LIN {X 0,Y 523.515,Z 618.573,A -85,B 0,C 180,E1 -4762.285,E2 -4762.285} C_VEL
LIN {X 0,Y 523.436,Z 624.082,A -85,B 0,C 180,E1 -4763.834,E2 -4763.834} C_VEL
LIN {X 0,Y 523.322,Z 628.245,A -85,B 0,C 180,E1 -4765.378,E2 -4765.378} C_VEL
LIN {X 0,Y 523.358,Z 631.166,A -85,B 0,C 180,E1 -4766.921,E2 -4766.921} C_VEL
LIN {X 0,Y 523.272,Z 632.904,A -85,B 0,C 180,E1 -4768.461,E2 -4768.461} C_VEL
LIN {X 0,Y 523.243,Z 633.498,A -85,B 0,C 180,E1 -4770,E2 -4770} C_VEL
LIN {X 0,Y 523.272,Z 632.901,A -85,B 0,C 180,E1 -4771.539,E2 -4771.539} C_VEL
LIN {X 0,Y 523.358,Z 631.161,A -85,B 0,C 180,E1 -4773.079,E2 -4773.079} C_VEL
LIN {X 0,Y 523.322,Z 628.242,A -85,B 0,C 180,E1 -4774.622,E2 -4774.622} C_VEL
LIN {X 0,Y 523.43,Z 624.086,A -85,B 0,C 180,E1 -4776.166,E2 -4776.166} C_VEL
LIN {X 0,Y 523.515,Z 618.574,A -85,B 0,C 180,E1 -4777.715,E2 -4777.715} C_VEL
LIN {X 0,Y 523.699,Z 611.561,A -85,B 0,C 180,E1 -4779.267,E2 -4779.267} C_VEL
LIN {X 0,Y 523.951,Z 602.835,A -85,B 0,C 180,E1 -4780.823,E2 -4780.823} C_VEL
LIN {X 0,Y 524.214,Z 593.543,A -85,B 0,C 180,E1 -4782.193,E2 -4782.193} C_VEL
LIN {X 0,Y 524.552,Z 584.141,A -85,B 0,C 180,E1 -4783.362,E2 -4783.362} C_VEL
LIN {X 0,Y 524.988,Z 571.926,A -85,B 0,C 180,E1 -4784.636,E2 -4784.636} C_VEL
LIN {X 0,Y 525.434,Z 560.572,A -85,B 0,C 180,E1 -4785.625,E2 -4785.625} C_VEL
LIN {X 0,Y 525.869,Z 547.217,A -85,B 0,C 180,E1 -4786.598,E2 -4786.598} C_VEL
LIN {X 0,Y 526.404,Z 533.994,A -85,B 0,C 180,E1 -4787.381,E2 -4787.381} C_VEL
LIN {X 0,Y 526.831,Z 519.537,A -85,B 0,C 180,E1 -4788.068,E2 -4788.068} C_VEL
LIN {X 0,Y 527.21,Z 505.352,A -85,B 0,C 180,E1 -4788.583,E2 -4788.583} C_VEL
LIN {X 0,Y 527.474,Z 490.49,A -85,B 0,C 180,E1 -4788.97,E2 -4788.97} C_VEL
LIN {X 0,Y 527.688,Z 469.477,A -85,B 0,C 180,E1 -4789.303,E2 -4789.303} C_VEL
LIN {X 0,Y 528.493,Z 334.8,A -85,B 0,C 180,E1 -4791.181,E2 -4791.181} C_VEL
LIN {X 0,Y 525.743,Z 320.905,A -85,B 0,C 180,E1 -4791.506,E2 -4791.506} C_VEL
LIN {X 0,Y 526.391,Z 301.543,A -85,B 0,C 180,E1 -4794.029,E2 -4794.029} C_VEL
LIN {X 0,Y 526.808,Z 285.78,A -85,B 0,C 180,E1 -4796.119,E2 -4796.119} C_VEL
LIN {X 0,Y 523.953,Z 272.848,A -85,B 0,C 180,E1 -4798.053,E2 -4798.053} C_VEL
LIN {X 0,Y 523.94,Z 272.843,A -85,B 0,C 180,E1 -4800.854,E2 -4800.854} C_VEL
LIN {X 0,Y 523.953,Z 272.844,A -85,B 0,C 180,E1 -4803.733,E2 -4803.733} C_VEL
LIN {X 0,Y 523.883,Z 272.854,A -85,B 0,C 180,E1 -4806.398,E2 -4806.398} C_VEL
LIN {X 0,Y 523.905,Z 272.847,A -85,B 0,C 180,E1 -4809.085,E2 -4809.085} C_VEL
LIN {X 0,Y 523.892,Z 272.856,A -85,B 0,C 180,E1 -4812.123,E2 -4812.123} C_VEL
LIN {X 0,Y 523.927,Z 272.844,A -85,B 0,C 180,E1 -4815.31,E2 -4815.31} C_VEL
LIN {X 0,Y 523.914,Z 272.845,A -85,B 0,C 180,E1 -4818.693,E2 -4818.693} C_VEL
LIN {X 0,Y 523.891,Z 272.854,A -85,B 0,C 180,E1 -4821.896,E2 -4821.896} C_VEL
LIN {X 0,Y 523.906,Z 272.844,A -85,B 0,C 180,E1 -4824.912,E2 -4824.912} C_VEL
LIN {X 0,Y 523.923,Z 272.849,A -85,B 0,C 180,E1 -4827.679,E2 -4827.679} C_VEL
LIN {X 0,Y 523.939,Z 272.841,A -85,B 0,C 180,E1 -4830.677,E2 -4830.677} C_VEL
LIN {X 0,Y 523.878,Z 272.856,A -85,B 0,C 180,E1 -4833.723,E2 -4833.723} C_VEL
LIN {X 0,Y 523.895,Z 272.848,A -85,B 0,C 180,E1 -4836.269,E2 -4836.269} C_VEL
LIN {X 0,Y 523.931,Z 272.842,A -85,B 0,C 180,E1 -4838.766,E2 -4838.766} C_VEL
LIN {X 0,Y 523.919,Z 272.84,A -85,B 0,C 180,E1 -4841.22,E2 -4841.22} C_VEL
LIN {X 0,Y 523.89,Z 272.855,A -85,B 0,C 180,E1 -4843.637,E2 -4843.637} C_VEL
LIN {X 0,Y 523.901,Z 272.846,A -85,B 0,C 180,E1 -4846.027,E2 -4846.027} C_VEL
LIN {X 0,Y 523.942,Z 272.83,A -85,B 0,C 180,E1 -4848.393,E2 -4848.393} C_VEL
LIN {X 0,Y 523.931,Z 272.85,A -85,B 0,C 180,E1 -4851.515,E2 -4851.515} C_VEL
LIN {X 0,Y 523.998,Z 272.835,A -85,B 0,C 180,E1 -4853.84,E2 -4853.84} C_VEL
LIN {X 0,Y 524.012,Z 272.835,A -85,B 0,C 180,E1 -4856.925,E2 -4856.925} C_VEL
LIN {X 0,Y 524.106,Z 272.825,A -85,B 0,C 180,E1 -4859.232,E2 -4859.232} C_VEL
LIN {X 0,Y 524.086,Z 272.821,A -85,B 0,C 180,E1 -4862.306,E2 -4862.306} C_VEL
LIN {X 0,Y 524.051,Z 272.834,A -85,B 0,C 180,E1 -4865.387,E2 -4865.387} C_VEL
LIN {X 0,Y 523.991,Z 272.838,A -85,B 0,C 180,E1 -4867.708,E2 -4867.708} C_VEL
LIN {X 0,Y 523.972,Z 272.839,A -85,B 0,C 180,E1 -4870.823,E2 -4870.823} C_VEL
LIN {X 0,Y 523.925,Z 272.852,A -85,B 0,C 180,E1 -4873.182,E2 -4873.182} C_VEL
LIN {X 0,Y 523.92,Z 272.847,A -85,B 0,C 180,E1 -4875.562,E2 -4875.562} C_VEL
LIN {X 0,Y 523.932,Z 272.841,A -85,B 0,C 180,E1 -4877.97,E2 -4877.97} C_VEL
LIN {X 0,Y 523.945,Z 272.834,A -85,B 0,C 180,E1 -4880.411,E2 -4880.411} C_VEL
LIN {X 0,Y 523.895,Z 272.85,A -85,B 0,C 180,E1 -4882.894,E2 -4882.894} C_VEL
LIN {X 0,Y 523.902,Z 272.847,A -85,B 0,C 180,E1 -4885.421,E2 -4885.421} C_VEL
LIN {X 0,Y 523.946,Z 272.835,A -85,B 0,C 180,E1 -4888,E2 -4888} C_VEL
LIN {X 0,Y 523.929,Z 272.85,A -85,B 0,C 180,E1 -4890.854,E2 -4890.854} C_VEL
LIN {X 0,Y 523.92,Z 272.844,A -85,B 0,C 180,E1 -4893.73,E2 -4893.73} C_VEL
LIN {X 0,Y 523.894,Z 272.849,A -85,B 0,C 180,E1 -4896.402,E2 -4896.402} C_VEL
LIN {X 0,Y 523.91,Z 272.849,A -85,B 0,C 180,E1 -4899.086,E2 -4899.086} C_VEL
LIN {X 0,Y 523.944,Z 272.841,A -85,B 0,C 180,E1 -4902.12,E2 -4902.12} C_VEL
LIN {X 0,Y 523.935,Z 272.844,A -85,B 0,C 180,E1 -4905.311,E2 -4905.311} C_VEL
LIN {X 0,Y 523.909,Z 272.852,A -85,B 0,C 180,E1 -4906.876,E2 -4906.876} C_VEL
LIN {X 0,Y 523.234,Z 272.932,A -85,B 0,C 180,E1 -4907.518,E2 -4907.518} C_VEL
LIN {X 0,Y 520.367,Z 273.294,A -85,B 0,C 180,E1 -4908.559,E2 -4908.559} C_VEL
LIN {X 0,Y 517.961,Z 273.589,A -85,B 0,C 180,E1 -4909.398,E2 -4909.398} C_VEL
LIN {X 0,Y 516.948,Z 273.715,A -85,B 0,C 180,E1 -4910.046,E2 -4910.046} C_VEL
LIN {X 0,Y 516.876,Z 273.725,A -85,B 0,C 180,E1 -4910.265,E2 -4910.265} C_VEL
LIN {X 0,Y 516.873,Z 273.722,A -85,B 0,C 180,E1 -4913.344,E2 -4913.344} C_VEL
LIN {X 0,Y 516.882,Z 273.724,A -85,B 0,C 180,E1 -4916.12,E2 -4916.12} C_VEL
LIN {X 0,Y 516.889,Z 273.725,A -85,B 0,C 180,E1 -4918.937,E2 -4918.937} C_VEL
LIN {X 0,Y 516.909,Z 273.72,A -85,B 0,C 180,E1 -4921.585,E2 -4921.585} C_VEL
LIN {X 0,Y 516.909,Z 273.725,A -85,B 0,C 180,E1 -4924.642,E2 -4924.642} C_VEL
LIN {X 0,Y 516.953,Z 273.863,A -85,B 0,C 180,E1 -4924.967,E2 -4924.967} C_VEL
LIN {X 0,Y 519.043,Z 283.843,A -85,B 0,C 180,E1 -4926.669,E2 -4926.669} C_VEL
LIN {X 0,Y 518.916,Z 294.305,A -85,B 0,C 180,E1 -4928.269,E2 -4928.269} C_VEL
LIN {X 0,Y 521.961,Z 307.972,A -85,B 0,C 180,E1 -4928.603,E2 -4928.603} C_VEL
LIN {X 0,Y 521.148,Z 429.496,A -85,B 0,C 180,E1 -4930.322,E2 -4930.322} C_VEL
LIN {X 0,Y 520.872,Z 460.237,A -85,B 0,C 180,E1 -4930.782,E2 -4930.782} C_VEL
LIN {X 0,Y 520.583,Z 475.638,A -85,B 0,C 180,E1 -4931.172,E2 -4931.172} C_VEL
LIN {X 0,Y 520.26,Z 490.103,A -85,B 0,C 180,E1 -4931.696,E2 -4931.696} C_VEL
LIN {X 0,Y 519.79,Z 502.789,A -85,B 0,C 180,E1 -4932.289,E2 -4932.289} C_VEL
LIN {X 0,Y 519.276,Z 516.39,A -85,B 0,C 180,E1 -4933.084,E2 -4933.084} C_VEL
LIN {X 0,Y 518.746,Z 529.412,A -85,B 0,C 180,E1 -4934.017,E2 -4934.017} C_VEL
LIN {X 0,Y 518.235,Z 541.543,A -85,B 0,C 180,E1 -4935.069,E2 -4935.069} C_VEL
LIN {X 0,Y 517.757,Z 553.011,A -85,B 0,C 180,E1 -4936.259,E2 -4936.259} C_VEL
LIN {X 0,Y 517.338,Z 562.659,A -85,B 0,C 180,E1 -4937.446,E2 -4937.446} C_VEL
LIN {X 0,Y 517.02,Z 572.112,A -85,B 0,C 180,E1 -4938.831,E2 -4938.831} C_VEL
LIN {X 0,Y 516.736,Z 579.983,A -85,B 0,C 180,E1 -4940.212,E2 -4940.212} C_VEL
LIN {X 0,Y 516.528,Z 587.329,A -85,B 0,C 180,E1 -4941.787,E2 -4941.787} C_VEL
LIN {X 0,Y 516.408,Z 591.836,A -85,B 0,C 180,E1 -4942.965,E2 -4942.965} C_VEL
LIN {X 0,Y 516.377,Z 596.61,A -85,B 0,C 180,E1 -4944.533,E2 -4944.533} C_VEL
LIN {X 0,Y 516.326,Z 600.112,A -85,B 0,C 180,E1 -4946.098,E2 -4946.098} C_VEL
LIN {X 0,Y 516.258,Z 602.432,A -85,B 0,C 180,E1 -4947.659,E2 -4947.659} C_VEL
LIN {X 0,Y 516.156,Z 603.623,A -85,B 0,C 180,E1 -4949.22,E2 -4949.22} C_VEL
LIN {X 0,Y 516.157,Z 603.642,A -85,B 0,C 180,E1 -4950.78,E2 -4950.78} C_VEL
LIN {X 0,Y 516.259,Z 602.527,A -85,B 0,C 180,E1 -4952.341,E2 -4952.341} C_VEL
LIN {X 0,Y 516.326,Z 600.282,A -85,B 0,C 180,E1 -4953.902,E2 -4953.902} C_VEL
LIN {X 0,Y 516.373,Z 596.852,A -85,B 0,C 180,E1 -4955.467,E2 -4955.467} C_VEL
LIN {X 0,Y 516.407,Z 592.155,A -85,B 0,C 180,E1 -4957.035,E2 -4957.035} C_VEL
LIN {X 0,Y 516.573,Z 586.066,A -85,B 0,C 180,E1 -4958.607,E2 -4958.607} C_VEL
LIN {X 0,Y 516.762,Z 578.399,A -85,B 0,C 180,E1 -4960.183,E2 -4960.183} C_VEL
LIN {X 0,Y 517.051,Z 570.22,A -85,B 0,C 180,E1 -4961.565,E2 -4961.565} C_VEL
LIN {X 0,Y 517.442,Z 560.368,A -85,B 0,C 180,E1 -4962.95,E2 -4962.95} C_VEL
LIN {X 0,Y 517.879,Z 550.263,A -85,B 0,C 180,E1 -4964.138,E2 -4964.138} C_VEL
LIN {X 0,Y 518.346,Z 538.482,A -85,B 0,C 180,E1 -4965.307,E2 -4965.307} C_VEL
LIN {X 0,Y 518.956,Z 525.014,A -85,B 0,C 180,E1 -4966.411,E2 -4966.411} C_VEL
LIN {X 0,Y 519.551,Z 511.488,A -85,B 0,C 180,E1 -4967.313,E2 -4967.313} C_VEL
LIN {X 0,Y 519.966,Z 497.613,A -85,B 0,C 180,E1 -4968.06,E2 -4968.06} C_VEL
LIN {X 0,Y 520.423,Z 483.39,A -85,B 0,C 180,E1 -4968.655,E2 -4968.655} C_VEL
LIN {X 0,Y 520.729,Z 468.583,A -85,B 0,C 180,E1 -4969.116,E2 -4969.116} C_VEL
LIN {X 0,Y 520.978,Z 453.076,A -85,B 0,C 180,E1 -4969.432,E2 -4969.432} C_VEL
LIN {X 0,Y 521.996,Z 308.384,A -85,B 0,C 180,E1 -4971.48,E2 -4971.48} C_VEL
LIN {X 0,Y 518.876,Z 293.935,A -85,B 0,C 180,E1 -4971.852,E2 -4971.852} C_VEL
LIN {X 0,Y 519.153,Z 284.409,A -85,B 0,C 180,E1 -4973.326,E2 -4973.326} C_VEL
LIN {X 0,Y 516.923,Z 273.723,A -85,B 0,C 180,E1 -4975.169,E2 -4975.169} C_VEL
LIN {X 0,Y 516.917,Z 273.723,A -85,B 0,C 180,E1 -4977.903,E2 -4977.903} C_VEL
LIN {X 0,Y 516.889,Z 273.723,A -85,B 0,C 180,E1 -4980.203,E2 -4980.203} C_VEL
LIN {X 0,Y 516.892,Z 273.724,A -85,B 0,C 180,E1 -4982.946,E2 -4982.946} C_VEL
LIN {X 0,Y 516.885,Z 273.727,A -85,B 0,C 180,E1 -4985.778,E2 -4985.778} C_VEL
LIN {X 0,Y 516.876,Z 273.725,A -85,B 0,C 180,E1 -4988.715,E2 -4988.715} C_VEL
LIN {X 0,Y 516.906,Z 273.722,A -85,B 0,C 180,E1 -4991.774,E2 -4991.774} C_VEL
LIN {X 0,Y 516.889,Z 273.725,A -85,B 0,C 180,E1 -4995.006,E2 -4995.006} C_VEL
LIN {X 0,Y 516.906,Z 273.712,A -85,B 0,C 180,E1 -4998.398,E2 -4998.398} C_VEL
LIN {X 0,Y 516.871,Z 273.728,A -85,B 0,C 180,E1 -5001.283,E2 -5001.283} C_VEL
LIN {X 0,Y 516.862,Z 273.719,A -85,B 0,C 180,E1 -5004.219,E2 -5004.219} C_VEL
LIN {X 0,Y 516.871,Z 273.729,A -85,B 0,C 180,E1 -5007.051,E2 -5007.051} C_VEL
LIN {X 0,Y 516.877,Z 273.716,A -85,B 0,C 180,E1 -5009.795,E2 -5009.795} C_VEL
LIN {X 0,Y 516.913,Z 273.718,A -85,B 0,C 180,E1 -5012.466,E2 -5012.466} C_VEL
LIN {X 0,Y 516.844,Z 273.732,A -85,B 0,C 180,E1 -5015.068,E2 -5015.068} C_VEL
LIN {X 0,Y 516.857,Z 273.723,A -85,B 0,C 180,E1 -5017.621,E2 -5017.621} C_VEL
LIN {X 0,Y 516.917,Z 273.716,A -85,B 0,C 180,E1 -5020.129,E2 -5020.129} C_VEL
LIN {X 0,Y 516.885,Z 273.722,A -85,B 0,C 180,E1 -5022.595,E2 -5022.595} C_VEL
LIN {X 0,Y 516.927,Z 273.72,A -85,B 0,C 180,E1 -5025.03,E2 -5025.03} C_VEL
LIN {X 0,Y 516.953,Z 273.712,A -85,B 0,C 180,E1 -5028.233,E2 -5028.233} C_VEL
LIN {X 0,Y 516.938,Z 273.713,A -85,B 0,C 180,E1 -5031.399,E2 -5031.399} C_VEL
LIN {X 0,Y 516.971,Z 273.709,A -85,B 0,C 180,E1 -5033.756,E2 -5033.756} C_VEL
LIN {X 0,Y 516.968,Z 273.716,A -85,B 0,C 180,E1 -5036.883,E2 -5036.883} C_VEL
LIN {X 0,Y 517.074,Z 273.696,A -85,B 0,C 180,E1 -5039.221,E2 -5039.221} C_VEL
LIN {X 0,Y 516.938,Z 273.713,A -85,B 0,C 180,E1 -5041.558,E2 -5041.558} C_VEL
LIN {X 0,Y 516.956,Z 273.713,A -85,B 0,C 180,E1 -5043.117,E2 -5043.117} C_VEL
LIN {X 0,Y 516.968,Z 273.713,A -85,B 0,C 180,E1 -5046.244,E2 -5046.244} C_VEL
LIN {X 0,Y 516.9,Z 273.716,A -85,B 0,C 180,E1 -5049.39,E2 -5049.39} C_VEL
LIN {X 0,Y 516.939,Z 273.715,A -85,B 0,C 180,E1 -5051.807,E2 -5051.807} C_VEL
LIN {X 0,Y 516.931,Z 273.716,A -85,B 0,C 180,E1 -5055.146,E2 -5055.146} C_VEL
LIN {X 0,Y 516.863,Z 273.727,A -85,B 0,C 180,E1 -5058.224,E2 -5058.224} C_VEL
LIN {X 0,Y 516.899,Z 273.722,A -85,B 0,C 180,E1 -5060.702,E2 -5060.702} C_VEL
LIN {X 0,Y 516.871,Z 273.728,A -85,B 0,C 180,E1 -5064.074,E2 -5064.074} C_VEL
LIN {X 0,Y 516.823,Z 273.732,A -85,B 0,C 180,E1 -5066.663,E2 -5066.663} C_VEL
LIN {X 0,Y 516.895,Z 273.72,A -85,B 0,C 180,E1 -5069.523,E2 -5069.523} C_VEL
LIN {X 0,Y 516.883,Z 273.722,A -85,B 0,C 180,E1 -5072.544,E2 -5072.544} C_VEL
LIN {X 0,Y 516.839,Z 273.726,A -85,B 0,C 180,E1 -5075.328,E2 -5075.328} C_VEL
LIN {X 0,Y 516.863,Z 273.723,A -85,B 0,C 180,E1 -5078.717,E2 -5078.717} C_VEL
LIN {X 0,Y 516.875,Z 273.721,A -85,B 0,C 180,E1 -5081.779,E2 -5081.779} C_VEL
LIN {X 0,Y 516.888,Z 273.72,A -85,B 0,C 180,E1 -5085.008,E2 -5085.008} C_VEL
LIN {X 0,Y 516.848,Z 273.728,A -85,B 0,C 180,E1 -5088.407,E2 -5088.407} C_VEL
LIN {X 0,Y 516.867,Z 273.724,A -85,B 0,C 180,E1 -5091.284,E2 -5091.284} C_VEL
LIN {X 0,Y 516.856,Z 273.726,A -85,B 0,C 180,E1 -5094.672,E2 -5094.672} C_VEL
LIN {X 0,Y 516.891,Z 273.725,A -85,B 0,C 180,E1 -5097.458,E2 -5097.458} C_VEL
LIN {X 0,Y 516.917,Z 273.721,A -85,B 0,C 180,E1 -5100.696,E2 -5100.696} C_VEL
LIN {X 0,Y 516.93,Z 273.878,A -85,B 0,C 180,E1 -5101.726,E2 -5101.726} C_VEL
LIN {X 0,Y 519.954,Z 287.167,A -85,B 0,C 180,E1 -5103.727,E2 -5103.727} C_VEL
LIN {X 0,Y 519.424,Z 306.078,A -85,B 0,C 180,E1 -5106.264,E2 -5106.264} C_VEL
LIN {X 0,Y 518.905,Z 320.752,A -85,B 0,C 180,E1 -5108.203,E2 -5108.203} C_VEL
LIN {X 0,Y 521.908,Z 336.644,A -85,B 0,C 180,E1 -5108.568,E2 -5108.568} C_VEL
LIN {X 0,Y 520.848,Z 486.861,A -85,B 0,C 180,E1 -5110.705,E2 -5110.705} C_VEL
LIN {X 0,Y 520.496,Z 502.829,A -85,B 0,C 180,E1 -5111.092,E2 -5111.092} C_VEL
LIN {X 0,Y 520.088,Z 518.191,A -85,B 0,C 180,E1 -5111.638,E2 -5111.638} C_VEL
LIN {X 0,Y 519.608,Z 531.979,A -85,B 0,C 180,E1 -5112.283,E2 -5112.283} C_VEL
LIN {X 0,Y 519.082,Z 545.494,A -85,B 0,C 180,E1 -5113.077,E2 -5113.077} C_VEL
LIN {X 0,Y 518.596,Z 558.466,A -85,B 0,C 180,E1 -5114.011,E2 -5114.011} C_VEL
LIN {X 0,Y 518.028,Z 571.715,A -85,B 0,C 180,E1 -5115.163,E2 -5115.163} C_VEL
LIN {X 0,Y 517.547,Z 583.935,A -85,B 0,C 180,E1 -5116.453,E2 -5116.453} C_VEL
LIN {X 0,Y 517.131,Z 594.805,A -85,B 0,C 180,E1 -5117.84,E2 -5117.84} C_VEL
LIN {X 0,Y 516.883,Z 603.856,A -85,B 0,C 180,E1 -5119.225,E2 -5119.225} C_VEL
LIN {X 0,Y 516.609,Z 611.362,A -85,B 0,C 180,E1 -5120.605,E2 -5120.605} C_VEL
LIN {X 0,Y 516.451,Z 618.369,A -85,B 0,C 180,E1 -5122.179,E2 -5122.179} C_VEL
LIN {X 0,Y 516.356,Z 623.878,A -85,B 0,C 180,E1 -5123.749,E2 -5123.749} C_VEL
LIN {X 0,Y 516.238,Z 628.041,A -85,B 0,C 180,E1 -5125.315,E2 -5125.315} C_VEL
LIN {X 0,Y 516.272,Z 630.963,A -85,B 0,C 180,E1 -5126.879,E2 -5126.879} C_VEL
LIN {X 0,Y 516.189,Z 632.703,A -85,B 0,C 180,E1 -5128.44,E2 -5128.44} C_VEL
LIN {X 0,Y 516.151,Z 633.299,A -85,B 0,C 180,E1 -5130,E2 -5130} C_VEL
LIN {X 0,Y 516.189,Z 632.7,A -85,B 0,C 180,E1 -5131.56,E2 -5131.56} C_VEL
LIN {X 0,Y 516.272,Z 630.958,A -85,B 0,C 180,E1 -5133.121,E2 -5133.121} C_VEL
LIN {X 0,Y 516.238,Z 628.039,A -85,B 0,C 180,E1 -5134.685,E2 -5134.685} C_VEL
LIN {X 0,Y 516.328,Z 623.881,A -85,B 0,C 180,E1 -5136.251,E2 -5136.251} C_VEL
LIN {X 0,Y 516.451,Z 618.37,A -85,B 0,C 180,E1 -5137.821,E2 -5137.821} C_VEL
LIN {X 0,Y 516.609,Z 611.356,A -85,B 0,C 180,E1 -5139.395,E2 -5139.395} C_VEL
LIN {X 0,Y 516.881,Z 603.852,A -85,B 0,C 180,E1 -5140.775,E2 -5140.775} C_VEL
LIN {X 0,Y 517.113,Z 595.075,A -85,B 0,C 180,E1 -5142.121,E2 -5142.121} C_VEL
LIN {X 0,Y 517.497,Z 585.575,A -85,B 0,C 180,E1 -5143.348,E2 -5143.348} C_VEL
LIN {X 0,Y 517.897,Z 574.703,A -85,B 0,C 180,E1 -5144.539,E2 -5144.539} C_VEL
LIN {X 0,Y 518.399,Z 563.427,A -85,B 0,C 180,E1 -5145.581,E2 -5145.581} C_VEL
LIN {X 0,Y 518.906,Z 549.877,A -85,B 0,C 180,E1 -5146.625,E2 -5146.625} C_VEL
LIN {X 0,Y 519.523,Z 535.561,A -85,B 0,C 180,E1 -5147.517,E2 -5147.517} C_VEL
LIN {X 0,Y 519.986,Z 521.595,A -85,B 0,C 180,E1 -5148.213,E2 -5148.213} C_VEL
LIN {X 0,Y 520.413,Z 506.675,A -85,B 0,C 180,E1 -5148.783,E2 -5148.783} C_VEL
LIN {X 0,Y 520.759,Z 491.492,A -85,B 0,C 180,E1 -5149.197,E2 -5149.197} C_VEL
LIN {X 0,Y 520.96,Z 472.786,A -85,B 0,C 180,E1 -5149.512,E2 -5149.512} C_VEL
LIN {X 0,Y 521.866,Z 335.88,A -85,B 0,C 180,E1 -5151.445,E2 -5151.445} C_VEL
LIN {X 0,Y 518.899,Z 320.738,A -85,B 0,C 180,E1 -5151.798,E2 -5151.798} C_VEL
LIN {X 0,Y 519.608,Z 299.781,A -85,B 0,C 180,E1 -5154.576,E2 -5154.576} C_VEL
LIN {X 0,Y 519.962,Z 287.167,A -85,B 0,C 180,E1 -5156.273,E2 -5156.273} C_VEL
LIN {X 0,Y 516.889,Z 273.728,A -85,B 0,C 180,E1 -5158.312,E2 -5158.312} C_VEL
LIN {X 0,Y 516.885,Z 273.721,A -85,B 0,C 180,E1 -5161.109,E2 -5161.109} C_VEL
LIN {X 0,Y 516.901,Z 273.724,A -85,B 0,C 180,E1 -5163.965,E2 -5163.965} C_VEL
LIN {X 0,Y 516.838,Z 273.729,A -85,B 0,C 180,E1 -5166.748,E2 -5166.748} C_VEL
LIN {X 0,Y 516.851,Z 273.73,A -85,B 0,C 180,E1 -5169.723,E2 -5169.723} C_VEL
LIN {X 0,Y 516.835,Z 273.728,A -85,B 0,C 180,E1 -5172.835,E2 -5172.835} C_VEL
LIN {X 0,Y 516.887,Z 273.72,A -85,B 0,C 180,E1 -5175.006,E2 -5175.006} C_VEL
LIN {X 0,Y 516.878,Z 273.724,A -85,B 0,C 180,E1 -5178.401,E2 -5178.401} C_VEL
LIN {X 0,Y 516.863,Z 273.724,A -85,B 0,C 180,E1 -5181.283,E2 -5181.283} C_VEL
LIN {X 0,Y 516.842,Z 273.725,A -85,B 0,C 180,E1 -5184.672,E2 -5184.672} C_VEL
LIN {X 0,Y 516.883,Z 273.723,A -85,B 0,C 180,E1 -5187.456,E2 -5187.456} C_VEL
LIN {X 0,Y 516.907,Z 273.717,A -85,B 0,C 180,E1 -5190.695,E2 -5190.695} C_VEL
LIN {X 0,Y 516.856,Z 273.732,A -85,B 0,C 180,E1 -5193.82,E2 -5193.82} C_VEL
LIN {X 0,Y 516.844,Z 273.724,A -85,B 0,C 180,E1 -5196.775,E2 -5196.775} C_VEL
LIN {X 0,Y 516.926,Z 273.716,A -85,B 0,C 180,E1 -5199.732,E2 -5199.732} C_VEL
LIN {X 0,Y 516.87,Z 273.719,A -85,B 0,C 180,E1 -5202.594,E2 -5202.594} C_VEL
LIN {X 0,Y 516.918,Z 273.718,A -85,B 0,C 180,E1 -5205.029,E2 -5205.029} C_VEL
LIN {X 0,Y 516.911,Z 273.706,A -85,B 0,C 180,E1 -5208.233,E2 -5208.233} C_VEL
LIN {X 0,Y 516.904,Z 273.723,A -85,B 0,C 180,E1 -5211.399,E2 -5211.399} C_VEL
LIN {X 0,Y 516.967,Z 273.712,A -85,B 0,C 180,E1 -5213.756,E2 -5213.756} C_VEL
LIN {X 0,Y 516.953,Z 273.714,A -85,B 0,C 180,E1 -5216.883,E2 -5216.883} C_VEL
LIN {X 0,Y 517.077,Z 273.7,A -85,B 0,C 180,E1 -5219.221,E2 -5219.221} C_VEL
LIN {X 0,Y 517.058,Z 273.696,A -85,B 0,C 180,E1 -5222.337,E2 -5222.337} C_VEL
LIN {X 0,Y 516.998,Z 273.711,A -85,B 0,C 180,E1 -5225.46,E2 -5225.46} C_VEL
LIN {X 0,Y 516.947,Z 273.714,A -85,B 0,C 180,E1 -5227.814,E2 -5227.814} C_VEL
LIN {X 0,Y 516.93,Z 273.718,A -85,B 0,C 180,E1 -5230.973,E2 -5230.973} C_VEL
LIN {X 0,Y 516.885,Z 273.726,A -85,B 0,C 180,E1 -5233.365,E2 -5233.365} C_VEL
LIN {X 0,Y 516.881,Z 273.722,A -85,B 0,C 180,E1 -5235.78,E2 -5235.78} C_VEL
LIN {X 0,Y 516.9,Z 273.717,A -85,B 0,C 180,E1 -5238.223,E2 -5238.223} C_VEL
LIN {X 0,Y 516.892,Z 273.715,A -85,B 0,C 180,E1 -5240.702,E2 -5240.702} C_VEL
LIN {X 0,Y 516.874,Z 273.721,A -85,B 0,C 180,E1 -5244.074,E2 -5244.074} C_VEL
LIN {X 0,Y 516.896,Z 273.72,A -85,B 0,C 180,E1 -5246.659,E2 -5246.659} C_VEL
LIN {X 0,Y 516.898,Z 273.72,A -85,B 0,C 180,E1 -5249.524,E2 -5249.524} C_VEL
LIN {X 0,Y 516.884,Z 273.722,A -85,B 0,C 180,E1 -5252.544,E2 -5252.544} C_VEL
LIN {X 0,Y 516.856,Z 273.726,A -85,B 0,C 180,E1 -5255.33,E2 -5255.33} C_VEL
LIN {X 0,Y 516.87,Z 273.721,A -85,B 0,C 180,E1 -5257.944,E2 -5257.944} C_VEL
LIN {X 0,Y 516.875,Z 273.727,A -85,B 0,C 180,E1 -5260.743,E2 -5260.743} C_VEL
LIN {X 0,Y 516.875,Z 273.728,A -85,B 0,C 180,E1 -5262.832,E2 -5262.832} C_VEL
LIN {X 0,Y 516.889,Z 273.726,A -85,B 0,C 180,E1 -5265.008,E2 -5265.008} C_VEL
LIN {X 0,Y 516.907,Z 273.722,A -85,B 0,C 180,E1 -5268.4,E2 -5268.4} C_VEL
LIN {X 0,Y 516.876,Z 273.725,A -85,B 0,C 180,E1 -5270.265,E2 -5270.265} C_VEL
LIN {X 0,Y 516.239,Z 273.809,A -85,B 0,C 180,E1 -5270.915,E2 -5270.915} C_VEL
LIN {X 0,Y 513.396,Z 274.163,A -85,B 0,C 180,E1 -5271.97,E2 -5271.97} C_VEL
LIN {X 0,Y 510.967,Z 274.464,A -85,B 0,C 180,E1 -5272.82,E2 -5272.82} C_VEL
LIN {X 0,Y 509.91,Z 274.59,A -85,B 0,C 180,E1 -5273.477,E2 -5273.477} C_VEL
LIN {X 0,Y 509.818,Z 274.6,A -85,B 0,C 180,E1 -5273.699,E2 -5273.699} C_VEL
LIN {X 0,Y 509.839,Z 274.603,A -85,B 0,C 180,E1 -5276.539,E2 -5276.539} C_VEL
LIN {X 0,Y 509.843,Z 274.6,A -85,B 0,C 180,E1 -5279.335,E2 -5279.335} C_VEL
LIN {X 0,Y 509.885,Z 274.598,A -85,B 0,C 180,E1 -5282.055,E2 -5282.055} C_VEL
LIN {X 0,Y 509.898,Z 274.718,A -85,B 0,C 180,E1 -5284.706,E2 -5284.706} C_VEL
LIN {X 0,Y 512.177,Z 285.37,A -85,B 0,C 180,E1 -5286.552,E2 -5286.552} C_VEL
LIN {X 0,Y 512.032,Z 294.252,A -85,B 0,C 180,E1 -5287.951,E2 -5287.951} C_VEL
LIN {X 0,Y 515.351,Z 308.882,A -85,B 0,C 180,E1 -5288.324,E2 -5288.324} C_VEL
LIN {X 0,Y 514.53,Z 420.915,A -85,B 0,C 180,E1 -5289.93,E2 -5289.93} C_VEL
LIN {X 0,Y 514.19,Z 460.064,A -85,B 0,C 180,E1 -5290.513,E2 -5290.513} C_VEL
LIN {X 0,Y 513.937,Z 475.097,A -85,B 0,C 180,E1 -5290.893,E2 -5290.893} C_VEL
LIN {X 0,Y 513.505,Z 490.321,A -85,B 0,C 180,E1 -5291.446,E2 -5291.446} C_VEL
LIN {X 0,Y 513.031,Z 503.004,A -85,B 0,C 180,E1 -5292.048,E2 -5292.048} C_VEL
LIN {X 0,Y 512.486,Z 516.603,A -85,B 0,C 180,E1 -5292.853,E2 -5292.853} C_VEL
LIN {X 0,Y 511.928,Z 529.234,A -85,B 0,C 180,E1 -5293.768,E2 -5293.768} C_VEL
LIN {X 0,Y 511.33,Z 541.754,A -85,B 0,C 180,E1 -5294.862,E2 -5294.862} C_VEL
LIN {X 0,Y 510.81,Z 553.221,A -85,B 0,C 180,E1 -5296.068,E2 -5296.068} C_VEL
LIN {X 0,Y 510.396,Z 562.868,A -85,B 0,C 180,E1 -5297.273,E2 -5297.273} C_VEL
LIN {X 0,Y 510.013,Z 572.392,A -85,B 0,C 180,E1 -5298.688,E2 -5298.688} C_VEL
LIN {X 0,Y 509.672,Z 581.19,A -85,B 0,C 180,E1 -5300.275,E2 -5300.275} C_VEL
LIN {X 0,Y 509.482,Z 587.535,A -85,B 0,C 180,E1 -5301.672,E2 -5301.672} C_VEL
LIN {X 0,Y 509.328,Z 593.488,A -85,B 0,C 180,E1 -5303.304,E2 -5303.304} C_VEL
LIN {X 0,Y 509.315,Z 596.815,A -85,B 0,C 180,E1 -5304.457,E2 -5304.457} C_VEL
LIN {X 0,Y 509.252,Z 600.316,A -85,B 0,C 180,E1 -5306.043,E2 -5306.043} C_VEL
LIN {X 0,Y 509.187,Z 602.635,A -85,B 0,C 180,E1 -5307.627,E2 -5307.627} C_VEL
LIN {X 0,Y 509.07,Z 603.825,A -85,B 0,C 180,E1 -5309.209,E2 -5309.209} C_VEL
LIN {X 0,Y 509.071,Z 603.844,A -85,B 0,C 180,E1 -5310.791,E2 -5310.791} C_VEL
LIN {X 0,Y 509.187,Z 602.729,A -85,B 0,C 180,E1 -5312.373,E2 -5312.373} C_VEL
LIN {X 0,Y 509.252,Z 600.484,A -85,B 0,C 180,E1 -5313.957,E2 -5313.957} C_VEL
LIN {X 0,Y 509.309,Z 597.053,A -85,B 0,C 180,E1 -5315.543,E2 -5315.543} C_VEL
LIN {X 0,Y 509.356,Z 592.356,A -85,B 0,C 180,E1 -5317.133,E2 -5317.133} C_VEL
LIN {X 0,Y 509.513,Z 586.267,A -85,B 0,C 180,E1 -5318.727,E2 -5318.727} C_VEL
LIN {X 0,Y 509.749,Z 578.599,A -85,B 0,C 180,E1 -5320.325,E2 -5320.325} C_VEL
LIN {X 0,Y 510.046,Z 570.08,A -85,B 0,C 180,E1 -5321.779,E2 -5321.779} C_VEL
LIN {X 0,Y 510.51,Z 560.567,A -85,B 0,C 180,E1 -5323.129,E2 -5323.129} C_VEL
LIN {X 0,Y 510.965,Z 550.461,A -85,B 0,C 180,E1 -5324.334,E2 -5324.334} C_VEL
LIN {X 0,Y 511.472,Z 538.907,A -85,B 0,C 180,E1 -5325.496,E2 -5325.496} C_VEL
LIN {X 0,Y 512.06,Z 526.624,A -85,B 0,C 180,E1 -5326.525,E2 -5326.525} C_VEL
LIN {X 0,Y 512.668,Z 513.259,A -85,B 0,C 180,E1 -5327.45,E2 -5327.45} C_VEL
LIN {X 0,Y 513.092,Z 500.777,A -85,B 0,C 180,E1 -5328.156,E2 -5328.156} C_VEL
LIN {X 0,Y 513.627,Z 486.172,A -85,B 0,C 180,E1 -5328.808,E2 -5328.808} C_VEL
LIN {X 0,Y 513.979,Z 471.261,A -85,B 0,C 180,E1 -5329.306,E2 -5329.306} C_VEL
LIN {X 0,Y 514.234,Z 456.861,A -85,B 0,C 180,E1 -5329.635,E2 -5329.635} C_VEL
LIN {X 0,Y 515.304,Z 318.846,A -85,B 0,C 180,E1 -5331.621,E2 -5331.621} C_VEL
LIN {X 0,Y 515.337,Z 308.907,A -85,B 0,C 180,E1 -5331.766,E2 -5331.766} C_VEL
LIN {X 0,Y 512.069,Z 294.209,A -85,B 0,C 180,E1 -5332.143,E2 -5332.143} C_VEL
LIN {X 0,Y 512.273,Z 285.925,A -85,B 0,C 180,E1 -5333.444,E2 -5333.444} C_VEL
LIN {X 0,Y 509.867,Z 274.603,A -85,B 0,C 180,E1 -5335.432,E2 -5335.432} C_VEL
LIN {X 0,Y 509.889,Z 274.597,A -85,B 0,C 180,E1 -5338.099,E2 -5338.099} C_VEL
LIN {X 0,Y 509.843,Z 274.606,A -85,B 0,C 180,E1 -5341.279,E2 -5341.279} C_VEL
LIN {X 0,Y 509.857,Z 274.598,A -85,B 0,C 180,E1 -5344.202,E2 -5344.202} C_VEL
LIN {X 0,Y 509.814,Z 274.608,A -85,B 0,C 180,E1 -5347.34,E2 -5347.34} C_VEL
LIN {X 0,Y 509.833,Z 274.596,A -85,B 0,C 180,E1 -5350.381,E2 -5350.381} C_VEL
LIN {X 0,Y 509.817,Z 274.607,A -85,B 0,C 180,E1 -5353.061,E2 -5353.061} C_VEL
LIN {X 0,Y 509.816,Z 274.603,A -85,B 0,C 180,E1 -5355.792,E2 -5355.792} C_VEL
LIN {X 0,Y 509.847,Z 274.592,A -85,B 0,C 180,E1 -5358.574,E2 -5358.574} C_VEL
LIN {X 0,Y 509.842,Z 274.597,A -85,B 0,C 180,E1 -5361.786,E2 -5361.786} C_VEL
LIN {X 0,Y 509.821,Z 274.598,A -85,B 0,C 180,E1 -5364.621,E2 -5364.621} C_VEL
LIN {X 0,Y 509.85,Z 274.597,A -85,B 0,C 180,E1 -5367.48,E2 -5367.48} C_VEL
LIN {X 0,Y 509.848,Z 274.591,A -85,B 0,C 180,E1 -5370.273,E2 -5370.273} C_VEL
LIN {X 0,Y 509.864,Z 274.602,A -85,B 0,C 180,E1 -5372.943,E2 -5372.943} C_VEL
LIN {X 0,Y 509.829,Z 274.601,A -85,B 0,C 180,E1 -5375.572,E2 -5375.572} C_VEL
LIN {X 0,Y 509.809,Z 274.6,A -85,B 0,C 180,E1 -5378.148,E2 -5378.148} C_VEL
LIN {X 0,Y 509.845,Z 274.602,A -85,B 0,C 180,E1 -5380.681,E2 -5380.681} C_VEL
LIN {X 0,Y 509.856,Z 274.6,A -85,B 0,C 180,E1 -5383.174,E2 -5383.174} C_VEL
LIN {X 0,Y 509.843,Z 274.596,A -85,B 0,C 180,E1 -5385.633,E2 -5385.633} C_VEL
LIN {X 0,Y 509.895,Z 274.599,A -85,B 0,C 180,E1 -5388.874,E2 -5388.874} C_VEL
LIN {X 0,Y 509.906,Z 274.589,A -85,B 0,C 180,E1 -5392.078,E2 -5392.078} C_VEL
LIN {X 0,Y 509.951,Z 274.589,A -85,B 0,C 180,E1 -5394.464,E2 -5394.464} C_VEL
LIN {X 0,Y 510.03,Z 274.574,A -85,B 0,C 180,E1 -5397.631,E2 -5397.631} C_VEL
LIN {X 0,Y 510.048,Z 274.578,A -85,B 0,C 180,E1 -5400.789,E2 -5400.789} C_VEL
LIN {X 0,Y 509.899,Z 274.591,A -85,B 0,C 180,E1 -5403.16,E2 -5403.16} C_VEL
LIN {X 0,Y 509.922,Z 274.592,A -85,B 0,C 180,E1 -5406.33,E2 -5406.33} C_VEL
LIN {X 0,Y 509.863,Z 274.598,A -85,B 0,C 180,E1 -5408.721,E2 -5408.721} C_VEL
LIN {X 0,Y 509.891,Z 274.594,A -85,B 0,C 180,E1 -5411.932,E2 -5411.932} C_VEL
LIN {X 0,Y 509.882,Z 274.594,A -85,B 0,C 180,E1 -5415.242,E2 -5415.242} C_VEL
LIN {X 0,Y 509.823,Z 274.607,A -85,B 0,C 180,E1 -5418.485,E2 -5418.485} C_VEL
LIN {X 0,Y 509.837,Z 274.599,A -85,B 0,C 180,E1 -5421.002,E2 -5421.002} C_VEL
LIN {X 0,Y 509.805,Z 274.603,A -85,B 0,C 180,E1 -5423.565,E2 -5423.565} C_VEL
LIN {X 0,Y 509.795,Z 274.609,A -85,B 0,C 180,E1 -5426.355,E2 -5426.355} C_VEL
LIN {X 0,Y 509.837,Z 274.6,A -85,B 0,C 180,E1 -5428.847,E2 -5428.847} C_VEL
LIN {X 0,Y 509.807,Z 274.603,A -85,B 0,C 180,E1 -5431.591,E2 -5431.591} C_VEL
LIN {X 0,Y 509.822,Z 274.606,A -85,B 0,C 180,E1 -5434.416,E2 -5434.416} C_VEL
LIN {X 0,Y 509.769,Z 274.606,A -85,B 0,C 180,E1 -5437.345,E2 -5437.345} C_VEL
LIN {X 0,Y 509.804,Z 274.6,A -85,B 0,C 180,E1 -5440.385,E2 -5440.385} C_VEL
LIN {X 0,Y 509.787,Z 274.605,A -85,B 0,C 180,E1 -5443.059,E2 -5443.059} C_VEL
LIN {X 0,Y 509.813,Z 274.607,A -85,B 0,C 180,E1 -5445.794,E2 -5445.794} C_VEL
LIN {X 0,Y 509.8,Z 274.605,A -85,B 0,C 180,E1 -5448.57,E2 -5448.57} C_VEL
LIN {X 0,Y 509.81,Z 274.607,A -85,B 0,C 180,E1 -5451.66,E2 -5451.66} C_VEL
LIN {X 0,Y 509.82,Z 274.603,A -85,B 0,C 180,E1 -5454.622,E2 -5454.622} C_VEL
LIN {X 0,Y 509.856,Z 274.602,A -85,B 0,C 180,E1 -5457.482,E2 -5457.482} C_VEL
LIN {X 0,Y 509.855,Z 274.603,A -85,B 0,C 180,E1 -5460.274,E2 -5460.274} C_VEL
LIN {X 0,Y 509.875,Z 274.722,A -85,B 0,C 180,E1 -5461.446,E2 -5461.446} C_VEL
LIN {X 0,Y 513.067,Z 288.554,A -85,B 0,C 180,E1 -5463.566,E2 -5463.566} C_VEL
LIN {X 0,Y 512.761,Z 301.167,A -85,B 0,C 180,E1 -5465.29,E2 -5465.29} C_VEL
LIN {X 0,Y 512.061,Z 320.577,A -85,B 0,C 180,E1 -5467.901,E2 -5467.901} C_VEL
LIN {X 0,Y 515.301,Z 337.748,A -85,B 0,C 180,E1 -5468.299,E2 -5468.299} C_VEL
LIN {X 0,Y 514.161,Z 486.89,A -85,B 0,C 180,E1 -5470.448,E2 -5470.448} C_VEL
LIN {X 0,Y 513.799,Z 502.627,A -85,B 0,C 180,E1 -5470.836,E2 -5470.836} C_VEL
LIN {X 0,Y 513.338,Z 517.987,A -85,B 0,C 180,E1 -5471.388,E2 -5471.388} C_VEL
LIN {X 0,Y 512.822,Z 531.775,A -85,B 0,C 180,E1 -5472.041,E2 -5472.041} C_VEL
LIN {X 0,Y 512.265,Z 545.29,A -85,B 0,C 180,E1 -5472.845,E2 -5472.845} C_VEL
LIN {X 0,Y 511.724,Z 557.755,A -85,B 0,C 180,E1 -5473.75,E2 -5473.75} C_VEL
LIN {X 0,Y 511.144,Z 570.435,A -85,B 0,C 180,E1 -5474.857,E2 -5474.857} C_VEL
LIN {X 0,Y 510.641,Z 581.958,A -85,B 0,C 180,E1 -5476.063,E2 -5476.063} C_VEL
LIN {X 0,Y 510.224,Z 591.658,A -85,B 0,C 180,E1 -5477.268,E2 -5477.268} C_VEL
LIN {X 0,Y 509.861,Z 601.343,A -85,B 0,C 180,E1 -5478.698,E2 -5478.698} C_VEL
LIN {X 0,Y 509.566,Z 609.126,A -85,B 0,C 180,E1 -5480.073,E2 -5480.073} C_VEL
LIN {X 0,Y 509.401,Z 616.541,A -85,B 0,C 180,E1 -5481.671,E2 -5481.671} C_VEL
LIN {X 0,Y 509.289,Z 622.423,A -85,B 0,C 180,E1 -5483.264,E2 -5483.264} C_VEL
LIN {X 0,Y 509.262,Z 625.919,A -85,B 0,C 180,E1 -5484.457,E2 -5484.457} C_VEL
LIN {X 0,Y 509.199,Z 629.451,A -85,B 0,C 180,E1 -5486.043,E2 -5486.043} C_VEL
LIN {X 0,Y 509.186,Z 631.775,A -85,B 0,C 180,E1 -5487.627,E2 -5487.627} C_VEL
LIN {X 0,Y 509.071,Z 632.942,A -85,B 0,C 180,E1 -5489.209,E2 -5489.209} C_VEL
LIN {X 0,Y 509.071,Z 632.941,A -85,B 0,C 180,E1 -5490.791,E2 -5490.791} C_VEL
LIN {X 0,Y 509.186,Z 631.771,A -85,B 0,C 180,E1 -5492.373,E2 -5492.373} C_VEL
LIN {X 0,Y 509.199,Z 629.446,A -85,B 0,C 180,E1 -5493.957,E2 -5493.957} C_VEL
LIN {X 0,Y 509.261,Z 625.92,A -85,B 0,C 180,E1 -5495.543,E2 -5495.543} C_VEL
LIN {X 0,Y 509.314,Z 621.1,A -85,B 0,C 180,E1 -5497.134,E2 -5497.134} C_VEL
LIN {X 0,Y 509.441,Z 614.857,A -85,B 0,C 180,E1 -5498.728,E2 -5498.728} C_VEL
LIN {X 0,Y 509.705,Z 607.02,A -85,B 0,C 180,E1 -5500.326,E2 -5500.326} C_VEL
LIN {X 0,Y 509.987,Z 598.429,A -85,B 0,C 180,E1 -5501.765,E2 -5501.765} C_VEL
LIN {X 0,Y 510.355,Z 588.643,A -85,B 0,C 180,E1 -5503.133,E2 -5503.133} C_VEL
LIN {X 0,Y 510.783,Z 578.374,A -85,B 0,C 180,E1 -5504.339,E2 -5504.339} C_VEL
LIN {X 0,Y 511.349,Z 566.95,A -85,B 0,C 180,E1 -5505.469,E2 -5505.469} C_VEL
LIN {X 0,Y 511.869,Z 553.873,A -85,B 0,C 180,E1 -5506.552,E2 -5506.552} C_VEL
LIN {X 0,Y 512.506,Z 540.525,A -85,B 0,C 180,E1 -5507.455,E2 -5507.455} C_VEL
LIN {X 0,Y 512.966,Z 527.786,A -85,B 0,C 180,E1 -5508.161,E2 -5508.161} C_VEL
LIN {X 0,Y 513.478,Z 512.888,A -85,B 0,C 180,E1 -5508.812,E2 -5508.812} C_VEL
LIN {X 0,Y 513.902,Z 497.582,A -85,B 0,C 180,E1 -5509.305,E2 -5509.305} C_VEL
LIN {X 0,Y 514.195,Z 481.956,A -85,B 0,C 180,E1 -5509.636,E2 -5509.636} C_VEL
LIN {X 0,Y 515.239,Z 336.875,A -85,B 0,C 180,E1 -5511.717,E2 -5511.717} C_VEL
LIN {X 0,Y 512.041,Z 320.369,A -85,B 0,C 180,E1 -5512.127,E2 -5512.127} C_VEL
LIN {X 0,Y 512.831,Z 299.59,A -85,B 0,C 180,E1 -5514.923,E2 -5514.923} C_VEL
LIN {X 0,Y 513.164,Z 290.134,A -85,B 0,C 180,E1 -5516.21,E2 -5516.21} C_VEL
LIN {X 0,Y 512.026,Z 283.79,A -85,B 0,C 180,E1 -5517.153,E2 -5517.153} C_VEL
LIN {X 0,Y 509.87,Z 274.6,A -85,B 0,C 180,E1 -5518.603,E2 -5518.603} C_VEL
LIN {X 0,Y 509.816,Z 274.604,A -85,B 0,C 180,E1 -5521.589,E2 -5521.589} C_VEL
LIN {X 0,Y 509.841,Z 274.603,A -85,B 0,C 180,E1 -5524.413,E2 -5524.413} C_VEL
LIN {X 0,Y 509.788,Z 274.606,A -85,B 0,C 180,E1 -5527.342,E2 -5527.342} C_VEL
LIN {X 0,Y 509.806,Z 274.608,A -85,B 0,C 180,E1 -5530.384,E2 -5530.384} C_VEL
LIN {X 0,Y 509.797,Z 274.607,A -85,B 0,C 180,E1 -5533.573,E2 -5533.573} C_VEL
LIN {X 0,Y 509.799,Z 274.606,A -85,B 0,C 180,E1 -5536.426,E2 -5536.426} C_VEL
LIN {X 0,Y 509.803,Z 274.604,A -85,B 0,C 180,E1 -5539.305,E2 -5539.305} C_VEL
LIN {X 0,Y 509.804,Z 274.609,A -85,B 0,C 180,E1 -5541.791,E2 -5541.791} C_VEL
LIN {X 0,Y 509.8,Z 274.602,A -85,B 0,C 180,E1 -5544.62,E2 -5544.62} C_VEL
LIN {X 0,Y 509.849,Z 274.599,A -85,B 0,C 180,E1 -5547.48,E2 -5547.48} C_VEL
LIN {X 0,Y 509.846,Z 274.599,A -85,B 0,C 180,E1 -5550.273,E2 -5550.273} C_VEL
LIN {X 0,Y 509.808,Z 274.6,A -85,B 0,C 180,E1 -5552.94,E2 -5552.94} C_VEL
LIN {X 0,Y 509.821,Z 274.607,A -85,B 0,C 180,E1 -5555.572,E2 -5555.572} C_VEL
LIN {X 0,Y 509.808,Z 274.603,A -85,B 0,C 180,E1 -5558.148,E2 -5558.148} C_VEL
LIN {X 0,Y 509.841,Z 274.59,A -85,B 0,C 180,E1 -5560.681,E2 -5560.681} C_VEL
LIN {X 0,Y 509.837,Z 274.598,A -85,B 0,C 180,E1 -5563.173,E2 -5563.173} C_VEL
LIN {X 0,Y 509.832,Z 274.604,A -85,B 0,C 180,E1 -5565.633,E2 -5565.633} C_VEL
LIN {X 0,Y 509.875,Z 274.582,A -85,B 0,C 180,E1 -5568.131,E2 -5568.131} C_VEL
LIN {X 0,Y 509.857,Z 274.598,A -85,B 0,C 180,E1 -5571.279,E2 -5571.279} C_VEL
LIN {X 0,Y 509.922,Z 274.59,A -85,B 0,C 180,E1 -5573.67,E2 -5573.67} C_VEL
LIN {X 0,Y 509.895,Z 274.592,A -85,B 0,C 180,E1 -5576.84,E2 -5576.84} C_VEL
LIN {X 0,Y 510.047,Z 274.575,A -85,B 0,C 180,E1 -5579.211,E2 -5579.211} C_VEL
LIN {X 0,Y 510.029,Z 274.572,A -85,B 0,C 180,E1 -5582.369,E2 -5582.369} C_VEL
LIN {X 0,Y 509.95,Z 274.588,A -85,B 0,C 180,E1 -5585.536,E2 -5585.536} C_VEL
LIN {X 0,Y 509.906,Z 274.59,A -85,B 0,C 180,E1 -5587.922,E2 -5587.922} C_VEL
LIN {X 0,Y 509.894,Z 274.596,A -85,B 0,C 180,E1 -5591.126,E2 -5591.126} C_VEL
LIN {X 0,Y 509.83,Z 274.598,A -85,B 0,C 180,E1 -5594.367,E2 -5594.367} C_VEL
LIN {X 0,Y 509.851,Z 274.6,A -85,B 0,C 180,E1 -5596.826,E2 -5596.826} C_VEL
LIN {X 0,Y 509.902,Z 274.581,A -85,B 0,C 180,E1 -5600.156,E2 -5600.156} C_VEL
LIN {X 0,Y 509.807,Z 274.604,A -85,B 0,C 180,E1 -5603.565,E2 -5603.565} C_VEL
LIN {X 0,Y 509.875,Z 274.591,A -85,B 0,C 180,E1 -5606.373,E2 -5606.373} C_VEL
LIN {X 0,Y 509.861,Z 274.596,A -85,B 0,C 180,E1 -5608.845,E2 -5608.845} C_VEL
LIN {X 0,Y 509.808,Z 274.601,A -85,B 0,C 180,E1 -5611.591,E2 -5611.591} C_VEL
LIN {X 0,Y 509.829,Z 274.601,A -85,B 0,C 180,E1 -5614.415,E2 -5614.415} C_VEL
LIN {X 0,Y 509.807,Z 274.603,A -85,B 0,C 180,E1 -5617.342,E2 -5617.342} C_VEL
LIN {X 0,Y 509.83,Z 274.6,A -85,B 0,C 180,E1 -5620.383,E2 -5620.383} C_VEL
LIN {X 0,Y 509.815,Z 274.606,A -85,B 0,C 180,E1 -5623.063,E2 -5623.063} C_VEL
LIN {X 0,Y 509.816,Z 274.601,A -85,B 0,C 180,E1 -5625.794,E2 -5625.794} C_VEL
LIN {X 0,Y 509.849,Z 274.604,A -85,B 0,C 180,E1 -5628.575,E2 -5628.575} C_VEL
LIN {X 0,Y 509.845,Z 274.596,A -85,B 0,C 180,E1 -5631.788,E2 -5631.788} C_VEL
LIN {X 0,Y 509.818,Z 274.6,A -85,B 0,C 180,E1 -5633.699,E2 -5633.699} C_VEL
LIN {X 0,Y 509.149,Z 274.687,A -85,B 0,C 180,E1 -5634.359,E2 -5634.359} C_VEL
LIN {X 0,Y 506.338,Z 275.039,A -85,B 0,C 180,E1 -5635.431,E2 -5635.431} C_VEL
LIN {X 0,Y 503.953,Z 275.338,A -85,B 0,C 180,E1 -5636.294,E2 -5636.294} C_VEL
LIN {X 0,Y 502.905,Z 275.467,A -85,B 0,C 180,E1 -5636.96,E2 -5636.96} C_VEL
LIN {X 0,Y 502.807,Z 275.477,A -85,B 0,C 180,E1 -5637.186,E2 -5637.186} C_VEL
LIN {X 0,Y 502.813,Z 275.478,A -85,B 0,C 180,E1 -5640.066,E2 -5640.066} C_VEL
LIN {X 0,Y 502.828,Z 275.471,A -85,B 0,C 180,E1 -5642.534,E2 -5642.534} C_VEL
LIN {X 0,Y 502.858,Z 275.566,A -85,B 0,C 180,E1 -5644.436,E2 -5644.436} C_VEL
LIN {X 0,Y 505.41,Z 287.926,A -85,B 0,C 180,E1 -5646.602,E2 -5646.602} C_VEL
LIN {X 0,Y 505.259,Z 294.447,A -85,B 0,C 180,E1 -5647.638,E2 -5647.638} C_VEL
LIN {X 0,Y 508.787,Z 310.772,A -85,B 0,C 180,E1 -5648.055,E2 -5648.055} C_VEL
LIN {X 0,Y 507.61,Z 456.857,A -85,B 0,C 180,E1 -5650.185,E2 -5650.185} C_VEL
LIN {X 0,Y 507.278,Z 471.999,A -85,B 0,C 180,E1 -5650.534,E2 -5650.534} C_VEL
LIN {X 0,Y 506.904,Z 486.743,A -85,B 0,C 180,E1 -5651.038,E2 -5651.038} C_VEL
LIN {X 0,Y 506.32,Z 501.242,A -85,B 0,C 180,E1 -5651.697,E2 -5651.697} C_VEL
LIN {X 0,Y 505.764,Z 515.24,A -85,B 0,C 180,E1 -5652.513,E2 -5652.513} C_VEL
LIN {X 0,Y 505.161,Z 528.033,A -85,B 0,C 180,E1 -5653.43,E2 -5653.43} C_VEL
LIN {X 0,Y 504.555,Z 540.189,A -85,B 0,C 180,E1 -5654.481,E2 -5654.481} C_VEL
LIN {X 0,Y 503.971,Z 551.66,A -85,B 0,C 180,E1 -5655.669,E2 -5655.669} C_VEL
LIN {X 0,Y 503.522,Z 561.601,A -85,B 0,C 180,E1 -5656.891,E2 -5656.891} C_VEL
LIN {X 0,Y 503.05,Z 571.308,A -85,B 0,C 180,E1 -5658.313,E2 -5658.313} C_VEL
LIN {X 0,Y 502.7,Z 579.396,A -85,B 0,C 180,E1 -5659.732,E2 -5659.732} C_VEL
LIN {X 0,Y 502.476,Z 586.066,A -85,B 0,C 180,E1 -5661.15,E2 -5661.15} C_VEL
LIN {X 0,Y 502.304,Z 592.246,A -85,B 0,C 180,E1 -5662.766,E2 -5662.766} C_VEL
LIN {X 0,Y 502.251,Z 597.019,A -85,B 0,C 180,E1 -5664.379,E2 -5664.379} C_VEL
LIN {X 0,Y 502.161,Z 600.52,A -85,B 0,C 180,E1 -5665.987,E2 -5665.987} C_VEL
LIN {X 0,Y 502.117,Z 602.838,A -85,B 0,C 180,E1 -5667.594,E2 -5667.594} C_VEL
LIN {X 0,Y 501.987,Z 604.028,A -85,B 0,C 180,E1 -5669.198,E2 -5669.198} C_VEL
LIN {X 0,Y 501.988,Z 604.047,A -85,B 0,C 180,E1 -5670.802,E2 -5670.802} C_VEL
LIN {X 0,Y 502.118,Z 602.931,A -85,B 0,C 180,E1 -5672.407,E2 -5672.407} C_VEL
LIN {X 0,Y 502.162,Z 600.686,A -85,B 0,C 180,E1 -5674.013,E2 -5674.013} C_VEL
LIN {X 0,Y 502.243,Z 597.254,A -85,B 0,C 180,E1 -5675.621,E2 -5675.621} C_VEL
LIN {X 0,Y 502.303,Z 592.557,A -85,B 0,C 180,E1 -5677.234,E2 -5677.234} C_VEL
LIN {X 0,Y 502.472,Z 586.468,A -85,B 0,C 180,E1 -5678.85,E2 -5678.85} C_VEL
LIN {X 0,Y 502.742,Z 578.799,A -85,B 0,C 180,E1 -5680.47,E2 -5680.47} C_VEL
LIN {X 0,Y 503.03,Z 570.67,A -85,B 0,C 180,E1 -5681.884,E2 -5681.884} C_VEL
LIN {X 0,Y 503.557,Z 560.766,A -85,B 0,C 180,E1 -5683.314,E2 -5683.314} C_VEL
LIN {X 0,Y 504.058,Z 550.66,A -85,B 0,C 180,E1 -5684.535,E2 -5684.535} C_VEL
LIN {X 0,Y 504.597,Z 539.408,A -85,B 0,C 180,E1 -5685.683,E2 -5685.683} C_VEL
LIN {X 0,Y 505.245,Z 526.563,A -85,B 0,C 180,E1 -5686.776,E2 -5686.776} C_VEL
LIN {X 0,Y 505.898,Z 513.452,A -85,B 0,C 180,E1 -5687.691,E2 -5687.691} C_VEL
LIN {X 0,Y 506.352,Z 500.968,A -85,B 0,C 180,E1 -5688.406,E2 -5688.406} C_VEL
LIN {X 0,Y 506.92,Z 486.645,A -85,B 0,C 180,E1 -5689.055,E2 -5689.055} C_VEL
LIN {X 0,Y 507.279,Z 471.558,A -85,B 0,C 180,E1 -5689.568,E2 -5689.568} C_VEL
LIN {X 0,Y 507.554,Z 457.026,A -85,B 0,C 180,E1 -5689.904,E2 -5689.904} C_VEL
LIN {X 0,Y 508.725,Z 319.129,A -85,B 0,C 180,E1 -5691.914,E2 -5691.914} C_VEL
LIN {X 0,Y 508.729,Z 310.004,A -85,B 0,C 180,E1 -5692.05,E2 -5692.05} C_VEL
LIN {X 0,Y 505.245,Z 294.406,A -85,B 0,C 180,E1 -5692.457,E2 -5692.457} C_VEL
LIN {X 0,Y 505.431,Z 287.726,A -85,B 0,C 180,E1 -5693.519,E2 -5693.519} C_VEL
LIN {X 0,Y 502.861,Z 275.476,A -85,B 0,C 180,E1 -5695.674,E2 -5695.674} C_VEL
LIN {X 0,Y 502.836,Z 275.474,A -85,B 0,C 180,E1 -5698.372,E2 -5698.372} C_VEL
LIN {X 0,Y 502.791,Z 275.485,A -85,B 0,C 180,E1 -5701.498,E2 -5701.498} C_VEL
LIN {X 0,Y 502.802,Z 275.476,A -85,B 0,C 180,E1 -5704.444,E2 -5704.444} C_VEL
LIN {X 0,Y 502.776,Z 275.484,A -85,B 0,C 180,E1 -5707.177,E2 -5707.177} C_VEL
LIN {X 0,Y 502.783,Z 275.476,A -85,B 0,C 180,E1 -5710.014,E2 -5710.014} C_VEL
LIN {X 0,Y 502.798,Z 275.477,A -85,B 0,C 180,E1 -5712.198,E2 -5712.198} C_VEL
LIN {X 0,Y 502.779,Z 275.484,A -85,B 0,C 180,E1 -5715.469,E2 -5715.469} C_VEL
LIN {X 0,Y 502.788,Z 275.471,A -85,B 0,C 180,E1 -5717.86,E2 -5717.86} C_VEL
LIN {X 0,Y 502.793,Z 275.482,A -85,B 0,C 180,E1 -5721.023,E2 -5721.023} C_VEL
LIN {X 0,Y 502.766,Z 275.475,A -85,B 0,C 180,E1 -5724.168,E2 -5724.168} C_VEL
LIN {X 0,Y 502.794,Z 275.483,A -85,B 0,C 180,E1 -5726.998,E2 -5726.998} C_VEL
LIN {X 0,Y 502.804,Z 275.468,A -85,B 0,C 180,E1 -5730.064,E2 -5730.064} C_VEL
LIN {X 0,Y 502.814,Z 275.475,A -85,B 0,C 180,E1 -5732.532,E2 -5732.532} C_VEL
LIN {X 0,Y 502.765,Z 275.484,A -85,B 0,C 180,E1 -5735.311,E2 -5735.311} C_VEL
LIN {X 0,Y 502.767,Z 275.477,A -85,B 0,C 180,E1 -5737.826,E2 -5737.826} C_VEL
LIN {X 0,Y 502.807,Z 275.476,A -85,B 0,C 180,E1 -5740.399,E2 -5740.399} C_VEL
LIN {X 0,Y 502.801,Z 275.48,A -85,B 0,C 180,E1 -5742.93,E2 -5742.93} C_VEL
LIN {X 0,Y 502.822,Z 275.472,A -85,B 0,C 180,E1 -5745.428,E2 -5745.428} C_VEL
LIN {X 0,Y 502.86,Z 275.474,A -85,B 0,C 180,E1 -5748.716,E2 -5748.716} C_VEL
LIN {X 0,Y 502.866,Z 275.465,A -85,B 0,C 180,E1 -5751.966,E2 -5751.966} C_VEL
LIN {X 0,Y 502.906,Z 275.465,A -85,B 0,C 180,E1 -5754.386,E2 -5754.386} C_VEL
LIN {X 0,Y 502.999,Z 275.45,A -85,B 0,C 180,E1 -5757.598,E2 -5757.598} C_VEL
LIN {X 0,Y 502.997,Z 275.456,A -85,B 0,C 180,E1 -5760.8,E2 -5760.8} C_VEL
LIN {X 0,Y 502.998,Z 275.455,A -85,B 0,C 180,E1 -5762.402,E2 -5762.402} C_VEL
LIN {X 0,Y 502.905,Z 275.46,A -85,B 0,C 180,E1 -5765.614,E2 -5765.614} C_VEL
LIN {X 0,Y 502.856,Z 275.47,A -85,B 0,C 180,E1 -5768.034,E2 -5768.034} C_VEL
LIN {X 0,Y 502.858,Z 275.469,A -85,B 0,C 180,E1 -5771.284,E2 -5771.284} C_VEL
LIN {X 0,Y 502.827,Z 275.479,A -85,B 0,C 180,E1 -5774.571,E2 -5774.571} C_VEL
LIN {X 0,Y 502.787,Z 275.477,A -85,B 0,C 180,E1 -5777.91,E2 -5777.91} C_VEL
LIN {X 0,Y 502.817,Z 275.478,A -85,B 0,C 180,E1 -5780.537,E2 -5780.537} C_VEL
LIN {X 0,Y 502.774,Z 275.479,A -85,B 0,C 180,E1 -5783.041,E2 -5783.041} C_VEL
LIN {X 0,Y 502.757,Z 275.481,A -85,B 0,C 180,E1 -5785.68,E2 -5785.68} C_VEL
LIN {X 0,Y 502.782,Z 275.484,A -85,B 0,C 180,E1 -5788.376,E2 -5788.376} C_VEL
LIN {X 0,Y 502.782,Z 275.477,A -85,B 0,C 180,E1 -5791.144,E2 -5791.144} C_VEL
LIN {X 0,Y 502.774,Z 275.481,A -85,B 0,C 180,E1 -5793.996,E2 -5793.996} C_VEL
LIN {X 0,Y 502.722,Z 275.484,A -85,B 0,C 180,E1 -5797.171,E2 -5797.171} C_VEL
LIN {X 0,Y 502.761,Z 275.479,A -85,B 0,C 180,E1 -5800.018,E2 -5800.018} C_VEL
LIN {X 0,Y 502.762,Z 275.485,A -85,B 0,C 180,E1 -5802.196,E2 -5802.196} C_VEL
LIN {X 0,Y 502.777,Z 275.48,A -85,B 0,C 180,E1 -5805.471,E2 -5805.471} C_VEL
LIN {X 0,Y 502.756,Z 275.48,A -85,B 0,C 180,E1 -5808.929,E2 -5808.929} C_VEL
LIN {X 0,Y 502.758,Z 275.487,A -85,B 0,C 180,E1 -5812.044,E2 -5812.044} C_VEL
LIN {X 0,Y 502.791,Z 275.478,A -85,B 0,C 180,E1 -5815.035,E2 -5815.035} C_VEL
LIN {X 0,Y 502.779,Z 275.485,A -85,B 0,C 180,E1 -5817.916,E2 -5817.916} C_VEL
LIN {X 0,Y 502.847,Z 275.561,A -85,B 0,C 180,E1 -5821.159,E2 -5821.159} C_VEL
LIN {X 0,Y 506.224,Z 290.209,A -85,B 0,C 180,E1 -5823.44,E2 -5823.44} C_VEL
LIN {X 0,Y 505.988,Z 301.012,A -85,B 0,C 180,E1 -5824.941,E2 -5824.941} C_VEL
LIN {X 0,Y 505.212,Z 320.313,A -85,B 0,C 180,E1 -5827.577,E2 -5827.577} C_VEL
LIN {X 0,Y 508.706,Z 338.569,A -85,B 0,C 180,E1 -5828.018,E2 -5828.018} C_VEL
LIN {X 0,Y 507.452,Z 486.686,A -85,B 0,C 180,E1 -5830.179,E2 -5830.179} C_VEL
LIN {X 0,Y 507.101,Z 502.424,A -85,B 0,C 180,E1 -5830.573,E2 -5830.573} C_VEL
LIN {X 0,Y 506.583,Z 517.968,A -85,B 0,C 180,E1 -5831.139,E2 -5831.139} C_VEL
LIN {X 0,Y 506.02,Z 531.571,A -85,B 0,C 180,E1 -5831.791,E2 -5831.791} C_VEL
LIN {X 0,Y 505.448,Z 545.086,A -85,B 0,C 180,E1 -5832.606,E2 -5832.606} C_VEL
LIN {X 0,Y 504.847,Z 557.55,A -85,B 0,C 180,E1 -5833.523,E2 -5833.523} C_VEL
LIN {X 0,Y 504.217,Z 570.23,A -85,B 0,C 180,E1 -5834.644,E2 -5834.644} C_VEL
LIN {X 0,Y 503.67,Z 581.752,A -85,B 0,C 180,E1 -5835.867,E2 -5835.867} C_VEL
LIN {X 0,Y 503.229,Z 591.453,A -85,B 0,C 180,E1 -5837.088,E2 -5837.088} C_VEL
LIN {X 0,Y 502.81,Z 601.148,A -85,B 0,C 180,E1 -5838.539,E2 -5838.539} C_VEL
LIN {X 0,Y 502.527,Z 608.922,A -85,B 0,C 180,E1 -5839.932,E2 -5839.932} C_VEL
LIN {X 0,Y 502.343,Z 616.336,A -85,B 0,C 180,E1 -5841.553,E2 -5841.553} C_VEL
LIN {X 0,Y 502.222,Z 622.22,A -85,B 0,C 180,E1 -5843.169,E2 -5843.169} C_VEL
LIN {X 0,Y 502.174,Z 625.715,A -85,B 0,C 180,E1 -5844.378,E2 -5844.378} C_VEL
LIN {X 0,Y 502.093,Z 629.247,A -85,B 0,C 180,E1 -5845.987,E2 -5845.987} C_VEL
LIN {X 0,Y 502.088,Z 631.572,A -85,B 0,C 180,E1 -5847.593,E2 -5847.593} C_VEL
LIN {X 0,Y 501.988,Z 632.739,A -85,B 0,C 180,E1 -5849.198,E2 -5849.198} C_VEL
LIN {X 0,Y 501.988,Z 632.739,A -85,B 0,C 180,E1 -5850.802,E2 -5850.802} C_VEL
LIN {X 0,Y 502.088,Z 631.568,A -85,B 0,C 180,E1 -5852.407,E2 -5852.407} C_VEL
LIN {X 0,Y 502.093,Z 629.243,A -85,B 0,C 180,E1 -5854.013,E2 -5854.013} C_VEL
LIN {X 0,Y 502.171,Z 625.716,A -85,B 0,C 180,E1 -5855.622,E2 -5855.622} C_VEL
LIN {X 0,Y 502.239,Z 620.896,A -85,B 0,C 180,E1 -5857.235,E2 -5857.235} C_VEL
LIN {X 0,Y 502.359,Z 614.652,A -85,B 0,C 180,E1 -5858.852,E2 -5858.852} C_VEL
LIN {X 0,Y 502.651,Z 606.815,A -85,B 0,C 180,E1 -5860.472,E2 -5860.472} C_VEL
LIN {X 0,Y 502.948,Z 597.78,A -85,B 0,C 180,E1 -5861.999,E2 -5861.999} C_VEL
LIN {X 0,Y 503.376,Z 588.438,A -85,B 0,C 180,E1 -5863.318,E2 -5863.318} C_VEL
LIN {X 0,Y 503.83,Z 578.169,A -85,B 0,C 180,E1 -5864.541,E2 -5864.541} C_VEL
LIN {X 0,Y 504.451,Z 565.941,A -85,B 0,C 180,E1 -5865.763,E2 -5865.763} C_VEL
LIN {X 0,Y 505.082,Z 552.332,A -85,B 0,C 180,E1 -5866.885,E2 -5866.885} C_VEL
LIN {X 0,Y 505.77,Z 538.694,A -85,B 0,C 180,E1 -5867.8,E2 -5867.8} C_VEL
LIN {X 0,Y 506.341,Z 524.57,A -85,B 0,C 180,E1 -5868.564,E2 -5868.564} C_VEL
LIN {X 0,Y 506.881,Z 509.415,A -85,B 0,C 180,E1 -5869.196,E2 -5869.196} C_VEL
LIN {X 0,Y 507.268,Z 494.166,A -85,B 0,C 180,E1 -5869.657,E2 -5869.657} C_VEL
LIN {X 0,Y 507.554,Z 478.289,A -85,B 0,C 180,E1 -5869.962,E2 -5869.962} C_VEL
LIN {X 0,Y 508.71,Z 338.79,A -85,B 0,C 180,E1 -5871.978,E2 -5871.978} C_VEL
LIN {X 0,Y 505.192,Z 320.339,A -85,B 0,C 180,E1 -5872.419,E2 -5872.419} C_VEL
LIN {X 0,Y 506.088,Z 298.778,A -85,B 0,C 180,E1 -5875.364,E2 -5875.364} C_VEL
LIN {X 0,Y 506.231,Z 290.202,A -85,B 0,C 180,E1 -5876.56,E2 -5876.56} C_VEL
LIN {X 0,Y 502.844,Z 275.474,A -85,B 0,C 180,E1 -5878.884,E2 -5878.884} C_VEL
LIN {X 0,Y 502.779,Z 275.479,A -85,B 0,C 180,E1 -5882.084,E2 -5882.084} C_VEL
LIN {X 0,Y 502.791,Z 275.477,A -85,B 0,C 180,E1 -5884.965,E2 -5884.965} C_VEL
LIN {X 0,Y 502.758,Z 275.485,A -85,B 0,C 180,E1 -5888.481,E2 -5888.481} C_VEL
LIN {X 0,Y 502.756,Z 275.482,A -85,B 0,C 180,E1 -5891.071,E2 -5891.071} C_VEL
LIN {X 0,Y 502.77,Z 275.483,A -85,B 0,C 180,E1 -5894.339,E2 -5894.339} C_VEL
LIN {X 0,Y 502.741,Z 275.483,A -85,B 0,C 180,E1 -5896.765,E2 -5896.765} C_VEL
LIN {X 0,Y 502.761,Z 275.48,A -85,B 0,C 180,E1 -5899.011,E2 -5899.011} C_VEL
LIN {X 0,Y 502.751,Z 275.487,A -85,B 0,C 180,E1 -5902.042,E2 -5902.042} C_VEL
LIN {X 0,Y 502.774,Z 275.477,A -85,B 0,C 180,E1 -5905.032,E2 -5905.032} C_VEL
LIN {X 0,Y 502.771,Z 275.486,A -85,B 0,C 180,E1 -5907.915,E2 -5907.915} C_VEL
LIN {X 0,Y 502.8,Z 275.474,A -85,B 0,C 180,E1 -5910.711,E2 -5910.711} C_VEL
LIN {X 0,Y 502.76,Z 275.483,A -85,B 0,C 180,E1 -5913.46,E2 -5913.46} C_VEL
LIN {X 0,Y 502.753,Z 275.483,A -85,B 0,C 180,E1 -5916.084,E2 -5916.084} C_VEL
LIN {X 0,Y 502.77,Z 275.478,A -85,B 0,C 180,E1 -5918.688,E2 -5918.688} C_VEL
LIN {X 0,Y 502.797,Z 275.47,A -85,B 0,C 180,E1 -5921.247,E2 -5921.247} C_VEL
LIN {X 0,Y 502.824,Z 275.472,A -85,B 0,C 180,E1 -5924.664,E2 -5924.664} C_VEL
LIN {X 0,Y 502.855,Z 275.457,A -85,B 0,C 180,E1 -5928.043,E2 -5928.043} C_VEL
LIN {X 0,Y 502.821,Z 275.473,A -85,B 0,C 180,E1 -5931.156,E2 -5931.156} C_VEL
LIN {X 0,Y 502.874,Z 275.469,A -85,B 0,C 180,E1 -5933.581,E2 -5933.581} C_VEL
LIN {X 0,Y 502.839,Z 275.471,A -85,B 0,C 180,E1 -5936.795,E2 -5936.795} C_VEL
LIN {X 0,Y 502.876,Z 275.462,A -85,B 0,C 180,E1 -5938.398,E2 -5938.398} C_VEL
LIN {X 0,Y 502.984,Z 275.453,A -85,B 0,C 180,E1 -5940,E2 -5940} C_VEL
LIN {X 0,Y 502.998,Z 275.448,A -85,B 0,C 180,E1 -5942.402,E2 -5942.402} C_VEL
LIN {X 0,Y 502.905,Z 275.464,A -85,B 0,C 180,E1 -5945.614,E2 -5945.614} C_VEL
LIN {X 0,Y 502.865,Z 275.467,A -85,B 0,C 180,E1 -5948.034,E2 -5948.034} C_VEL
LIN {X 0,Y 502.86,Z 275.473,A -85,B 0,C 180,E1 -5951.284,E2 -5951.284} C_VEL
LIN {X 0,Y 502.812,Z 275.473,A -85,B 0,C 180,E1 -5954.572,E2 -5954.572} C_VEL
LIN {X 0,Y 502.798,Z 275.482,A -85,B 0,C 180,E1 -5957.07,E2 -5957.07} C_VEL
LIN {X 0,Y 502.806,Z 275.467,A -85,B 0,C 180,E1 -5959.601,E2 -5959.601} C_VEL
LIN {X 0,Y 502.79,Z 275.476,A -85,B 0,C 180,E1 -5962.702,E2 -5962.702} C_VEL
LIN {X 0,Y 502.785,Z 275.474,A -85,B 0,C 180,E1 -5965.679,E2 -5965.679} C_VEL
LIN {X 0,Y 502.826,Z 275.466,A -85,B 0,C 180,E1 -5968.374,E2 -5968.374} C_VEL
LIN {X 0,Y 502.782,Z 275.477,A -85,B 0,C 180,E1 -5971.499,E2 -5971.499} C_VEL
LIN {X 0,Y 502.782,Z 275.479,A -85,B 0,C 180,E1 -5974.443,E2 -5974.443} C_VEL
LIN {X 0,Y 502.768,Z 275.482,A -85,B 0,C 180,E1 -5977.178,E2 -5977.178} C_VEL
LIN {X 0,Y 502.78,Z 275.476,A -85,B 0,C 180,E1 -5980.016,E2 -5980.016} C_VEL
LIN {X 0,Y 502.796,Z 275.476,A -85,B 0,C 180,E1 -5982.2,E2 -5982.2} C_VEL
LIN {X 0,Y 502.779,Z 275.479,A -85,B 0,C 180,E1 -5985.471,E2 -5985.471} C_VEL
LIN {X 0,Y 502.814,Z 275.48,A -85,B 0,C 180,E1 -5988.935,E2 -5988.935} C_VEL
LIN {X 0,Y 502.788,Z 275.476,A -85,B 0,C 180,E1 -5992.047,E2 -5992.047} C_VEL
LIN {X 0,Y 502.793,Z 275.481,A -85,B 0,C 180,E1 -5995.035,E2 -5995.035} C_VEL
LIN {X 0,Y 502.807,Z 275.477,A -85,B 0,C 180,E1 -5997.186,E2 -5997.186} C_VEL
LIN {X 0,Y 502.104,Z 275.565,A -85,B 0,C 180,E1 -5997.854,E2 -5997.854} C_VEL
LIN {X 0,Y 499.241,Z 275.923,A -85,B 0,C 180,E1 -5998.94,E2 -5998.94} C_VEL
LIN {X 0,Y 496.847,Z 276.222,A -85,B 0,C 180,E1 -5999.815,E2 -5999.815} C_VEL
LIN {X 0,Y 495.829,Z 276.349,A -85,B 0,C 180,E1 -6000.491,E2 -6000.491} C_VEL
LIN {X 0,Y 495.749,Z 276.357,A -85,B 0,C 180,E1 -6000.719,E2 -6000.719} C_VEL
LIN {X 0,Y 495.802,Z 276.35,A -85,B 0,C 180,E1 -6003.934,E2 -6003.934} C_VEL
LIN {X 0,Y 495.841,Z 276.431,A -85,B 0,C 180,E1 -6004.162,E2 -6004.162} C_VEL
LIN {X 0,Y 498.508,Z 288.998,A -85,B 0,C 180,E1 -6006.402,E2 -6006.402} C_VEL
LIN {X 0,Y 498.453,Z 294.645,A -85,B 0,C 180,E1 -6007.316,E2 -6007.316} C_VEL
LIN {X 0,Y 502.197,Z 311.108,A -85,B 0,C 180,E1 -6007.753,E2 -6007.753} C_VEL
LIN {X 0,Y 500.956,Z 457.094,A -85,B 0,C 180,E1 -6009.911,E2 -6009.911} C_VEL
LIN {X 0,Y 500.616,Z 472.162,A -85,B 0,C 180,E1 -6010.263,E2 -6010.263} C_VEL
LIN {X 0,Y 500.204,Z 487.021,A -85,B 0,C 180,E1 -6010.777,E2 -6010.777} C_VEL
LIN {X 0,Y 499.568,Z 501.458,A -85,B 0,C 180,E1 -6011.441,E2 -6011.441} C_VEL
LIN {X 0,Y 498.983,Z 515.453,A -85,B 0,C 180,E1 -6012.268,E2 -6012.268} C_VEL
LIN {X 0,Y 498.34,Z 528.24,A -85,B 0,C 180,E1 -6013.196,E2 -6013.196} C_VEL
LIN {X 0,Y 497.678,Z 540.522,A -85,B 0,C 180,E1 -6014.273,E2 -6014.273} C_VEL
LIN {X 0,Y 497.077,Z 551.869,A -85,B 0,C 180,E1 -6015.466,E2 -6015.466} C_VEL
LIN {X 0,Y 496.558,Z 561.81,A -85,B 0,C 180,E1 -6016.704,E2 -6016.704} C_VEL
LIN {X 0,Y 496.049,Z 570.675,A -85,B 0,C 180,E1 -6018.005,E2 -6018.005} C_VEL
LIN {X 0,Y 495.749,Z 578.51,A -85,B 0,C 180,E1 -6019.38,E2 -6019.38} C_VEL
LIN {X 0,Y 495.446,Z 586.273,A -85,B 0,C 180,E1 -6021.023,E2 -6021.023} C_VEL
LIN {X 0,Y 495.242,Z 592.452,A -85,B 0,C 180,E1 -6022.662,E2 -6022.662} C_VEL
LIN {X 0,Y 495.186,Z 597.224,A -85,B 0,C 180,E1 -6024.299,E2 -6024.299} C_VEL
LIN {X 0,Y 495.061,Z 600.725,A -85,B 0,C 180,E1 -6025.93,E2 -6025.93} C_VEL
LIN {X 0,Y 495.021,Z 603.042,A -85,B 0,C 180,E1 -6027.559,E2 -6027.559} C_VEL
LIN {X 0,Y 494.907,Z 604.231,A -85,B 0,C 180,E1 -6029.186,E2 -6029.186} C_VEL
LIN {X 0,Y 494.908,Z 604.249,A -85,B 0,C 180,E1 -6030.814,E2 -6030.814} C_VEL
LIN {X 0,Y 495.022,Z 603.133,A -85,B 0,C 180,E1 -6032.441,E2 -6032.441} C_VEL
LIN {X 0,Y 495.06,Z 600.888,A -85,B 0,C 180,E1 -6034.07,E2 -6034.07} C_VEL
LIN {X 0,Y 495.177,Z 597.456,A -85,B 0,C 180,E1 -6035.702,E2 -6035.702} C_VEL
LIN {X 0,Y 495.242,Z 592.758,A -85,B 0,C 180,E1 -6037.338,E2 -6037.338} C_VEL
LIN {X 0,Y 495.44,Z 586.669,A -85,B 0,C 180,E1 -6038.977,E2 -6038.977} C_VEL
LIN {X 0,Y 495.743,Z 578.999,A -85,B 0,C 180,E1 -6040.62,E2 -6040.62} C_VEL
LIN {X 0,Y 496.115,Z 570.003,A -85,B 0,C 180,E1 -6042.188,E2 -6042.188} C_VEL
LIN {X 0,Y 496.614,Z 560.965,A -85,B 0,C 180,E1 -6043.503,E2 -6043.503} C_VEL
LIN {X 0,Y 497.144,Z 550.858,A -85,B 0,C 180,E1 -6044.741,E2 -6044.741} C_VEL
LIN {X 0,Y 497.738,Z 539.877,A -85,B 0,C 180,E1 -6045.878,E2 -6045.878} C_VEL
LIN {X 0,Y 498.366,Z 528.043,A -85,B 0,C 180,E1 -6046.909,E2 -6046.909} C_VEL
LIN {X 0,Y 499.058,Z 515.22,A -85,B 0,C 180,E1 -6047.836,E2 -6047.836} C_VEL
LIN {X 0,Y 499.627,Z 501.158,A -85,B 0,C 180,E1 -6048.663,E2 -6048.663} C_VEL
LIN {X 0,Y 500.245,Z 486.048,A -85,B 0,C 180,E1 -6049.351,E2 -6049.351} C_VEL
LIN {X 0,Y 500.604,Z 471.219,A -85,B 0,C 180,E1 -6049.855,E2 -6049.855} C_VEL
LIN {X 0,Y 500.912,Z 456.912,A -85,B 0,C 180,E1 -6050.185,E2 -6050.185} C_VEL
LIN {X 0,Y 502.151,Z 319.296,A -85,B 0,C 180,E1 -6052.216,E2 -6052.216} C_VEL
LIN {X 0,Y 502.206,Z 311.215,A -85,B 0,C 180,E1 -6052.336,E2 -6052.336} C_VEL
LIN {X 0,Y 498.434,Z 294.616,A -85,B 0,C 180,E1 -6052.779,E2 -6052.779} C_VEL
LIN {X 0,Y 498.578,Z 289.419,A -85,B 0,C 180,E1 -6053.616,E2 -6053.616} C_VEL
LIN {X 0,Y 495.818,Z 276.351,A -85,B 0,C 180,E1 -6055.952,E2 -6055.952} C_VEL
LIN {X 0,Y 495.768,Z 276.355,A -85,B 0,C 180,E1 -6058.814,E2 -6058.814} C_VEL
LIN {X 0,Y 495.753,Z 276.359,A -85,B 0,C 180,E1 -6061.724,E2 -6061.724} C_VEL
LIN {X 0,Y 495.772,Z 276.353,A -85,B 0,C 180,E1 -6064.694,E2 -6064.694} C_VEL
LIN {X 0,Y 495.727,Z 276.363,A -85,B 0,C 180,E1 -6067.561,E2 -6067.561} C_VEL
LIN {X 0,Y 495.761,Z 276.35,A -85,B 0,C 180,E1 -6070.699,E2 -6070.699} C_VEL
LIN {X 0,Y 495.722,Z 276.358,A -85,B 0,C 180,E1 -6074.001,E2 -6074.001} C_VEL
LIN {X 0,Y 495.718,Z 276.362,A -85,B 0,C 180,E1 -6077.116,E2 -6077.116} C_VEL
LIN {X 0,Y 495.748,Z 276.354,A -85,B 0,C 180,E1 -6080.361,E2 -6080.361} C_VEL
LIN {X 0,Y 495.719,Z 276.356,A -85,B 0,C 180,E1 -6083.455,E2 -6083.455} C_VEL
LIN {X 0,Y 495.733,Z 276.356,A -85,B 0,C 180,E1 -6086.434,E2 -6086.434} C_VEL
LIN {X 0,Y 495.74,Z 276.35,A -85,B 0,C 180,E1 -6089.312,E2 -6089.312} C_VEL
LIN {X 0,Y 495.765,Z 276.351,A -85,B 0,C 180,E1 -6092.108,E2 -6092.108} C_VEL
LIN {X 0,Y 495.723,Z 276.36,A -85,B 0,C 180,E1 -6094.829,E2 -6094.829} C_VEL
LIN {X 0,Y 495.736,Z 276.355,A -85,B 0,C 180,E1 -6097.494,E2 -6097.494} C_VEL
LIN {X 0,Y 495.755,Z 276.353,A -85,B 0,C 180,E1 -6100.109,E2 -6100.109} C_VEL
LIN {X 0,Y 495.746,Z 276.356,A -85,B 0,C 180,E1 -6102.68,E2 -6102.68} C_VEL
LIN {X 0,Y 495.771,Z 276.353,A -85,B 0,C 180,E1 -6105.216,E2 -6105.216} C_VEL
LIN {X 0,Y 495.836,Z 276.346,A -85,B 0,C 180,E1 -6108.554,E2 -6108.554} C_VEL
LIN {X 0,Y 495.822,Z 276.342,A -85,B 0,C 180,E1 -6111.851,E2 -6111.851} C_VEL
LIN {X 0,Y 495.862,Z 276.342,A -85,B 0,C 180,E1 -6114.306,E2 -6114.306} C_VEL
LIN {X 0,Y 495.968,Z 276.326,A -85,B 0,C 180,E1 -6117.563,E2 -6117.563} C_VEL
LIN {X 0,Y 495.948,Z 276.334,A -85,B 0,C 180,E1 -6120.812,E2 -6120.812} C_VEL
LIN {X 0,Y 495.966,Z 276.332,A -85,B 0,C 180,E1 -6122.436,E2 -6122.436} C_VEL
LIN {X 0,Y 495.861,Z 276.338,A -85,B 0,C 180,E1 -6125.694,E2 -6125.694} C_VEL
LIN {X 0,Y 495.813,Z 276.348,A -85,B 0,C 180,E1 -6128.149,E2 -6128.149} C_VEL
LIN {X 0,Y 495.834,Z 276.343,A -85,B 0,C 180,E1 -6131.445,E2 -6131.445} C_VEL
LIN {X 0,Y 495.773,Z 276.355,A -85,B 0,C 180,E1 -6134.783,E2 -6134.783} C_VEL
LIN {X 0,Y 495.767,Z 276.354,A -85,B 0,C 180,E1 -6138.172,E2 -6138.172} C_VEL
LIN {X 0,Y 495.762,Z 276.354,A -85,B 0,C 180,E1 -6140.757,E2 -6140.757} C_VEL
LIN {X 0,Y 495.726,Z 276.357,A -85,B 0,C 180,E1 -6143.388,E2 -6143.388} C_VEL
LIN {X 0,Y 495.726,Z 276.359,A -85,B 0,C 180,E1 -6146.73,E2 -6146.73} C_VEL
LIN {X 0,Y 495.751,Z 276.356,A -85,B 0,C 180,E1 -6149.747,E2 -6149.747} C_VEL
LIN {X 0,Y 495.741,Z 276.354,A -85,B 0,C 180,E1 -6152.596,E2 -6152.596} C_VEL
LIN {X 0,Y 495.717,Z 276.359,A -85,B 0,C 180,E1 -6155.54,E2 -6155.54} C_VEL
LIN {X 0,Y 495.73,Z 276.355,A -85,B 0,C 180,E1 -6158.765,E2 -6158.765} C_VEL
LIN {X 0,Y 495.735,Z 276.353,A -85,B 0,C 180,E1 -6161.783,E2 -6161.783} C_VEL
LIN {X 0,Y 495.729,Z 276.357,A -85,B 0,C 180,E1 -6165.142,E2 -6165.142} C_VEL
LIN {X 0,Y 495.716,Z 276.362,A -85,B 0,C 180,E1 -6168.216,E2 -6168.216} C_VEL
LIN {X 0,Y 495.734,Z 276.356,A -85,B 0,C 180,E1 -6171.236,E2 -6171.236} C_VEL
LIN {X 0,Y 495.738,Z 276.358,A -85,B 0,C 180,E1 -6174.463,E2 -6174.463} C_VEL
LIN {X 0,Y 495.763,Z 276.357,A -85,B 0,C 180,E1 -6177.406,E2 -6177.406} C_VEL
LIN {X 0,Y 495.789,Z 276.354,A -85,B 0,C 180,E1 -6180.839,E2 -6180.839} C_VEL
LIN {X 0,Y 499.288,Z 291.326,A -85,B 0,C 180,E1 -6183.229,E2 -6183.229} C_VEL
LIN {X 0,Y 499.399,Z 296.058,A -85,B 0,C 180,E1 -6183.911,E2 -6183.911} C_VEL
LIN {X 0,Y 498.548,Z 316.487,A -85,B 0,C 180,E1 -6186.753,E2 -6186.753} C_VEL
LIN {X 0,Y 498.342,Z 320.091,A -85,B 0,C 180,E1 -6187.249,E2 -6187.249} C_VEL
LIN {X 0,Y 502.059,Z 338.901,A -85,B 0,C 180,E1 -6187.72,E2 -6187.72} C_VEL
LIN {X 0,Y 500.877,Z 479.891,A -85,B 0,C 180,E1 -6189.79,E2 -6189.79} C_VEL
LIN {X 0,Y 500.546,Z 495.424,A -85,B 0,C 180,E1 -6190.108,E2 -6190.108} C_VEL
LIN {X 0,Y 500.133,Z 509.873,A -85,B 0,C 180,E1 -6190.56,E2 -6190.56} C_VEL
LIN {X 0,Y 499.603,Z 524.366,A -85,B 0,C 180,E1 -6191.176,E2 -6191.176} C_VEL
LIN {X 0,Y 498.928,Z 538.496,A -85,B 0,C 180,E1 -6191.948,E2 -6191.948} C_VEL
LIN {X 0,Y 498.236,Z 552.122,A -85,B 0,C 180,E1 -6192.875,E2 -6192.875} C_VEL
LIN {X 0,Y 497.553,Z 565.437,A -85,B 0,C 180,E1 -6193.985,E2 -6193.985} C_VEL
LIN {X 0,Y 496.859,Z 577.961,A -85,B 0,C 180,E1 -6195.25,E2 -6195.25} C_VEL
LIN {X 0,Y 496.399,Z 588.232,A -85,B 0,C 180,E1 -6196.491,E2 -6196.491} C_VEL
LIN {X 0,Y 495.878,Z 598.305,A -85,B 0,C 180,E1 -6197.939,E2 -6197.939} C_VEL
LIN {X 0,Y 495.613,Z 606.616,A -85,B 0,C 180,E1 -6199.377,E2 -6199.377} C_VEL
LIN {X 0,Y 495.29,Z 614.451,A -85,B 0,C 180,E1 -6201.02,E2 -6201.02} C_VEL
LIN {X 0,Y 495.159,Z 620.688,A -85,B 0,C 180,E1 -6202.661,E2 -6202.661} C_VEL
LIN {X 0,Y 495.068,Z 625.511,A -85,B 0,C 180,E1 -6204.297,E2 -6204.297} C_VEL
LIN {X 0,Y 494.99,Z 629.044,A -85,B 0,C 180,E1 -6205.929,E2 -6205.929} C_VEL
LIN {X 0,Y 494.994,Z 631.369,A -85,B 0,C 180,E1 -6207.559,E2 -6207.559} C_VEL
LIN {X 0,Y 494.908,Z 632.537,A -85,B 0,C 180,E1 -6209.186,E2 -6209.186} C_VEL
LIN {X 0,Y 494.908,Z 632.536,A -85,B 0,C 180,E1 -6210.814,E2 -6210.814} C_VEL
LIN {X 0,Y 494.994,Z 631.365,A -85,B 0,C 180,E1 -6212.441,E2 -6212.441} C_VEL
LIN {X 0,Y 494.99,Z 629.039,A -85,B 0,C 180,E1 -6214.071,E2 -6214.071} C_VEL
LIN {X 0,Y 495.066,Z 625.512,A -85,B 0,C 180,E1 -6215.703,E2 -6215.703} C_VEL
LIN {X 0,Y 495.159,Z 620.692,A -85,B 0,C 180,E1 -6217.339,E2 -6217.339} C_VEL
LIN {X 0,Y 495.29,Z 614.448,A -85,B 0,C 180,E1 -6218.98,E2 -6218.98} C_VEL
LIN {X 0,Y 495.613,Z 606.61,A -85,B 0,C 180,E1 -6220.623,E2 -6220.623} C_VEL
LIN {X 0,Y 495.898,Z 598.232,A -85,B 0,C 180,E1 -6222.072,E2 -6222.072} C_VEL
LIN {X 0,Y 496.399,Z 588.233,A -85,B 0,C 180,E1 -6223.509,E2 -6223.509} C_VEL
LIN {X 0,Y 496.883,Z 577.964,A -85,B 0,C 180,E1 -6224.749,E2 -6224.749} C_VEL
LIN {X 0,Y 497.565,Z 565.389,A -85,B 0,C 180,E1 -6226.02,E2 -6226.02} C_VEL
LIN {X 0,Y 498.232,Z 552.128,A -85,B 0,C 180,E1 -6227.125,E2 -6227.125} C_VEL
LIN {X 0,Y 498.986,Z 538.49,A -85,B 0,C 180,E1 -6228.05,E2 -6228.05} C_VEL
LIN {X 0,Y 499.594,Z 524.367,A -85,B 0,C 180,E1 -6228.824,E2 -6228.824} C_VEL
LIN {X 0,Y 500.13,Z 510.043,A -85,B 0,C 180,E1 -6229.434,E2 -6229.434} C_VEL
LIN {X 0,Y 500.54,Z 494.864,A -85,B 0,C 180,E1 -6229.909,E2 -6229.909} C_VEL
LIN {X 0,Y 500.888,Z 479.053,A -85,B 0,C 180,E1 -6230.225,E2 -6230.225} C_VEL
LIN {X 0,Y 502.056,Z 338.946,A -85,B 0,C 180,E1 -6232.28,E2 -6232.28} C_VEL
LIN {X 0,Y 498.339,Z 320.136,A -85,B 0,C 180,E1 -6232.744,E2 -6232.744} C_VEL
LIN {X 0,Y 499.3,Z 299.566,A -85,B 0,C 180,E1 -6235.595,E2 -6235.595} C_VEL
LIN {X 0,Y 499.5,Z 292.902,A -85,B 0,C 180,E1 -6236.533,E2 -6236.533} C_VEL
LIN {X 0,Y 496.812,Z 280.622,A -85,B 0,C 180,E1 -6238.456,E2 -6238.456} C_VEL
LIN {X 0,Y 495.789,Z 276.352,A -85,B 0,C 180,E1 -6239.161,E2 -6239.161} C_VEL
LIN {X 0,Y 495.763,Z 276.354,A -85,B 0,C 180,E1 -6242.594,E2 -6242.594} C_VEL
LIN {X 0,Y 495.738,Z 276.357,A -85,B 0,C 180,E1 -6245.537,E2 -6245.537} C_VEL
LIN {X 0,Y 495.734,Z 276.358,A -85,B 0,C 180,E1 -6248.764,E2 -6248.764} C_VEL
LIN {X 0,Y 495.716,Z 276.363,A -85,B 0,C 180,E1 -6251.784,E2 -6251.784} C_VEL
LIN {X 0,Y 495.729,Z 276.357,A -85,B 0,C 180,E1 -6255.14,E2 -6255.14} C_VEL
LIN {X 0,Y 495.734,Z 276.36,A -85,B 0,C 180,E1 -6258.217,E2 -6258.217} C_VEL
LIN {X 0,Y 495.73,Z 276.357,A -85,B 0,C 180,E1 -6261.235,E2 -6261.235} C_VEL
LIN {X 0,Y 495.72,Z 276.357,A -85,B 0,C 180,E1 -6264.46,E2 -6264.46} C_VEL
LIN {X 0,Y 495.741,Z 276.356,A -85,B 0,C 180,E1 -6267.404,E2 -6267.404} C_VEL
LIN {X 0,Y 495.75,Z 276.355,A -85,B 0,C 180,E1 -6270.253,E2 -6270.253} C_VEL
LIN {X 0,Y 495.726,Z 276.357,A -85,B 0,C 180,E1 -6273.27,E2 -6273.27} C_VEL
LIN {X 0,Y 495.726,Z 276.355,A -85,B 0,C 180,E1 -6276.612,E2 -6276.612} C_VEL
LIN {X 0,Y 495.767,Z 276.354,A -85,B 0,C 180,E1 -6279.324,E2 -6279.324} C_VEL
LIN {X 0,Y 495.766,Z 276.35,A -85,B 0,C 180,E1 -6281.828,E2 -6281.828} C_VEL
LIN {X 0,Y 495.763,Z 276.355,A -85,B 0,C 180,E1 -6285.216,E2 -6285.216} C_VEL
LIN {X 0,Y 495.805,Z 276.332,A -85,B 0,C 180,E1 -6288.554,E2 -6288.554} C_VEL
LIN {X 0,Y 495.801,Z 276.35,A -85,B 0,C 180,E1 -6291.851,E2 -6291.851} C_VEL
LIN {X 0,Y 495.861,Z 276.336,A -85,B 0,C 180,E1 -6294.306,E2 -6294.306} C_VEL
LIN {X 0,Y 495.965,Z 276.33,A -85,B 0,C 180,E1 -6297.564,E2 -6297.564} C_VEL
LIN {X 0,Y 495.954,Z 276.329,A -85,B 0,C 180,E1 -6300,E2 -6300} C_VEL
LIN {X 0,Y 495.967,Z 276.323,A -85,B 0,C 180,E1 -6302.437,E2 -6302.437} C_VEL
LIN {X 0,Y 495.862,Z 276.341,A -85,B 0,C 180,E1 -6305.694,E2 -6305.694} C_VEL
LIN {X 0,Y 495.821,Z 276.344,A -85,B 0,C 180,E1 -6308.149,E2 -6308.149} C_VEL
LIN {X 0,Y 495.835,Z 276.348,A -85,B 0,C 180,E1 -6311.446,E2 -6311.446} C_VEL
LIN {X 0,Y 495.763,Z 276.353,A -85,B 0,C 180,E1 -6314.784,E2 -6314.784} C_VEL
LIN {X 0,Y 495.744,Z 276.359,A -85,B 0,C 180,E1 -6317.32,E2 -6317.32} C_VEL
LIN {X 0,Y 495.754,Z 276.343,A -85,B 0,C 180,E1 -6319.891,E2 -6319.891} C_VEL
LIN {X 0,Y 495.746,Z 276.355,A -85,B 0,C 180,E1 -6322.861,E2 -6322.861} C_VEL
LIN {X 0,Y 495.748,Z 276.35,A -85,B 0,C 180,E1 -6326.07,E2 -6326.07} C_VEL
LIN {X 0,Y 495.759,Z 276.351,A -85,B 0,C 180,E1 -6328.816,E2 -6328.816} C_VEL
LIN {X 0,Y 495.744,Z 276.352,A -85,B 0,C 180,E1 -6331.726,E2 -6331.726} C_VEL
LIN {X 0,Y 495.753,Z 276.358,A -85,B 0,C 180,E1 -6334.694,E2 -6334.694} C_VEL
LIN {X 0,Y 495.72,Z 276.356,A -85,B 0,C 180,E1 -6337.563,E2 -6337.563} C_VEL
LIN {X 0,Y 495.758,Z 276.357,A -85,B 0,C 180,E1 -6340.701,E2 -6340.701} C_VEL
LIN {X 0,Y 495.721,Z 276.357,A -85,B 0,C 180,E1 -6344.003,E2 -6344.003} C_VEL
LIN {X 0,Y 495.72,Z 276.362,A -85,B 0,C 180,E1 -6347.118,E2 -6347.118} C_VEL
LIN {X 0,Y 495.753,Z 276.354,A -85,B 0,C 180,E1 -6349.954,E2 -6349.954} C_VEL
LIN {X 0,Y 495.723,Z 276.362,A -85,B 0,C 180,E1 -6352.554,E2 -6352.554} C_VEL
LIN {X 0,Y 495.768,Z 276.353,A -85,B 0,C 180,E1 -6355.457,E2 -6355.457} C_VEL
LIN {X 0,Y 495.752,Z 276.36,A -85,B 0,C 180,E1 -6358.365,E2 -6358.365} C_VEL
LIN {X 0,Y 495.749,Z 276.357,A -85,B 0,C 180,E1 -6360.719,E2 -6360.719} C_VEL
LIN {X 0,Y 495.093,Z 276.44,A -85,B 0,C 180,E1 -6361.172,E2 -6361.172} C_VEL
LIN {X 0,Y 492.307,Z 276.787,A -85,B 0,C 180,E1 -6361.882,E2 -6361.882} C_VEL
LIN {X 0,Y 489.484,Z 277.132,A -85,B 0,C 180,E1 -6362.599,E2 -6362.599} C_VEL
LIN {X 0,Y 488.79,Z 277.216,A -85,B 0,C 180,E1 -6363.061,E2 -6363.061} C_VEL
LIN {X 0,Y 488.767,Z 277.293,A -85,B 0,C 180,E1 -6363.874,E2 -6363.874} C_VEL
LIN {X 0,Y 491.562,Z 290.168,A -85,B 0,C 180,E1 -6366.21,E2 -6366.21} C_VEL
LIN {X 0,Y 491.612,Z 294.857,A -85,B 0,C 180,E1 -6366.983,E2 -6366.983} C_VEL
LIN {X 0,Y 495.656,Z 312.503,A -85,B 0,C 180,E1 -6367.461,E2 -6367.461} C_VEL
LIN {X 0,Y 494.315,Z 457.325,A -85,B 0,C 180,E1 -6369.629,E2 -6369.629} C_VEL
LIN {X 0,Y 493.968,Z 471.314,A -85,B 0,C 180,E1 -6369.954,E2 -6369.954} C_VEL
LIN {X 0,Y 493.562,Z 486.233,A -85,B 0,C 180,E1 -6370.466,E2 -6370.466} C_VEL
LIN {X 0,Y 492.857,Z 501.671,A -85,B 0,C 180,E1 -6371.179,E2 -6371.179} C_VEL
LIN {X 0,Y 492.222,Z 515.665,A -85,B 0,C 180,E1 -6372.016,E2 -6372.016} C_VEL
LIN {X 0,Y 491.535,Z 528.451,A -85,B 0,C 180,E1 -6372.956,E2 -6372.956} C_VEL
LIN {X 0,Y 490.802,Z 540.86,A -85,B 0,C 180,E1 -6374.06,E2 -6374.06} C_VEL
LIN {X 0,Y 490.172,Z 552.078,A -85,B 0,C 180,E1 -6375.257,E2 -6375.257} C_VEL
LIN {X 0,Y 489.633,Z 562.018,A -85,B 0,C 180,E1 -6376.512,E2 -6376.512} C_VEL
LIN {X 0,Y 489.04,Z 571.351,A -85,B 0,C 180,E1 -6377.908,E2 -6377.908} C_VEL
LIN {X 0,Y 488.671,Z 579.81,A -85,B 0,C 180,E1 -6379.434,E2 -6379.434} C_VEL
LIN {X 0,Y 488.405,Z 586.479,A -85,B 0,C 180,E1 -6380.893,E2 -6380.893} C_VEL
LIN {X 0,Y 488.176,Z 592.658,A -85,B 0,C 180,E1 -6382.556,E2 -6382.556} C_VEL
LIN {X 0,Y 488.1,Z 597.429,A -85,B 0,C 180,E1 -6384.215,E2 -6384.215} C_VEL
LIN {X 0,Y 487.962,Z 600.93,A -85,B 0,C 180,E1 -6385.87,E2 -6385.87} C_VEL
LIN {X 0,Y 487.929,Z 603.245,A -85,B 0,C 180,E1 -6387.523,E2 -6387.523} C_VEL
LIN {X 0,Y 487.831,Z 604.433,A -85,B 0,C 180,E1 -6389.175,E2 -6389.175} C_VEL
LIN {X 0,Y 487.831,Z 604.451,A -85,B 0,C 180,E1 -6390.825,E2 -6390.825} C_VEL
LIN {X 0,Y 487.93,Z 603.336,A -85,B 0,C 180,E1 -6392.477,E2 -6392.477} C_VEL
LIN {X 0,Y 487.961,Z 601.091,A -85,B 0,C 180,E1 -6394.13,E2 -6394.13} C_VEL
LIN {X 0,Y 488.092,Z 597.657,A -85,B 0,C 180,E1 -6395.785,E2 -6395.785} C_VEL
LIN {X 0,Y 488.175,Z 592.96,A -85,B 0,C 180,E1 -6397.444,E2 -6397.444} C_VEL
LIN {X 0,Y 488.396,Z 586.87,A -85,B 0,C 180,E1 -6399.107,E2 -6399.107} C_VEL
LIN {X 0,Y 488.751,Z 579.199,A -85,B 0,C 180,E1 -6400.774,E2 -6400.774} C_VEL
LIN {X 0,Y 489.134,Z 570.609,A -85,B 0,C 180,E1 -6402.301,E2 -6402.301} C_VEL
LIN {X 0,Y 489.671,Z 561.164,A -85,B 0,C 180,E1 -6403.698,E2 -6403.698} C_VEL
LIN {X 0,Y 490.243,Z 551.057,A -85,B 0,C 180,E1 -6404.954,E2 -6404.954} C_VEL
LIN {X 0,Y 490.881,Z 540.32,A -85,B 0,C 180,E1 -6406.081,E2 -6406.081} C_VEL
LIN {X 0,Y 491.547,Z 528.24,A -85,B 0,C 180,E1 -6407.15,E2 -6407.15} C_VEL
LIN {X 0,Y 492.289,Z 515.415,A -85,B 0,C 180,E1 -6408.089,E2 -6408.089} C_VEL
LIN {X 0,Y 492.914,Z 501.351,A -85,B 0,C 180,E1 -6408.927,E2 -6408.927} C_VEL
LIN {X 0,Y 493.551,Z 486.622,A -85,B 0,C 180,E1 -6409.608,E2 -6409.608} C_VEL
LIN {X 0,Y 493.935,Z 471.948,A -85,B 0,C 180,E1 -6410.118,E2 -6410.118} C_VEL
LIN {X 0,Y 494.256,Z 457.367,A -85,B 0,C 180,E1 -6410.463,E2 -6410.463} C_VEL
LIN {X 0,Y 495.544,Z 325.675,A -85,B 0,C 180,E1 -6412.433,E2 -6412.433} C_VEL
LIN {X 0,Y 495.517,Z 311.685,A -85,B 0,C 180,E1 -6412.649,E2 -6412.649} C_VEL
LIN {X 0,Y 491.652,Z 294.821,A -85,B 0,C 180,E1 -6413.11,E2 -6413.11} C_VEL
LIN {X 0,Y 491.652,Z 290.55,A -85,B 0,C 180,E1 -6413.814,E2 -6413.814} C_VEL
LIN {X 0,Y 488.756,Z 277.229,A -85,B 0,C 180,E1 -6416.241,E2 -6416.241} C_VEL
LIN {X 0,Y 488.72,Z 277.236,A -85,B 0,C 180,E1 -6419.27,E2 -6419.27} C_VEL
LIN {X 0,Y 488.7,Z 277.235,A -85,B 0,C 180,E1 -6422.146,E2 -6422.146} C_VEL
LIN {X 0,Y 488.719,Z 277.234,A -85,B 0,C 180,E1 -6425.114,E2 -6425.114} C_VEL
LIN {X 0,Y 488.676,Z 277.238,A -85,B 0,C 180,E1 -6428.199,E2 -6428.199} C_VEL
LIN {X 0,Y 488.714,Z 277.227,A -85,B 0,C 180,E1 -6430.344,E2 -6430.344} C_VEL
LIN {X 0,Y 488.678,Z 277.239,A -85,B 0,C 180,E1 -6433.654,E2 -6433.654} C_VEL
LIN {X 0,Y 488.677,Z 277.235,A -85,B 0,C 180,E1 -6436.344,E2 -6436.344} C_VEL
LIN {X 0,Y 488.696,Z 277.235,A -85,B 0,C 180,E1 -6439.673,E2 -6439.673} C_VEL
LIN {X 0,Y 488.67,Z 277.235,A -85,B 0,C 180,E1 -6442.84,E2 -6442.84} C_VEL
LIN {X 0,Y 488.712,Z 277.231,A -85,B 0,C 180,E1 -6445.886,E2 -6445.886} C_VEL
LIN {X 0,Y 488.681,Z 277.231,A -85,B 0,C 180,E1 -6448.819,E2 -6448.819} C_VEL
LIN {X 0,Y 488.731,Z 277.229,A -85,B 0,C 180,E1 -6451.67,E2 -6451.67} C_VEL
LIN {X 0,Y 488.699,Z 277.231,A -85,B 0,C 180,E1 -6454.441,E2 -6454.441} C_VEL
LIN {X 0,Y 488.709,Z 277.234,A -85,B 0,C 180,E1 -6457.152,E2 -6457.152} C_VEL
LIN {X 0,Y 488.711,Z 277.23,A -85,B 0,C 180,E1 -6459.81,E2 -6459.81} C_VEL
LIN {X 0,Y 488.698,Z 277.231,A -85,B 0,C 180,E1 -6462.422,E2 -6462.422} C_VEL
LIN {X 0,Y 488.745,Z 277.231,A -85,B 0,C 180,E1 -6464.999,E2 -6464.999} C_VEL
LIN {X 0,Y 488.791,Z 277.222,A -85,B 0,C 180,E1 -6468.387,E2 -6468.387} C_VEL
LIN {X 0,Y 488.77,Z 277.221,A -85,B 0,C 180,E1 -6471.733,E2 -6471.733} C_VEL
LIN {X 0,Y 488.822,Z 277.218,A -85,B 0,C 180,E1 -6474.224,E2 -6474.224} C_VEL
LIN {X 0,Y 488.936,Z 277.202,A -85,B 0,C 180,E1 -6477.528,E2 -6477.528} C_VEL
LIN {X 0,Y 488.9,Z 277.212,A -85,B 0,C 180,E1 -6480.824,E2 -6480.824} C_VEL
LIN {X 0,Y 488.933,Z 277.208,A -85,B 0,C 180,E1 -6482.471,E2 -6482.471} C_VEL
LIN {X 0,Y 488.82,Z 277.215,A -85,B 0,C 180,E1 -6485.776,E2 -6485.776} C_VEL
LIN {X 0,Y 488.758,Z 277.229,A -85,B 0,C 180,E1 -6488.267,E2 -6488.267} C_VEL
LIN {X 0,Y 488.79,Z 277.221,A -85,B 0,C 180,E1 -6491.613,E2 -6491.613} C_VEL
LIN {X 0,Y 488.747,Z 277.228,A -85,B 0,C 180,E1 -6495.001,E2 -6495.001} C_VEL
LIN {X 0,Y 488.732,Z 277.233,A -85,B 0,C 180,E1 -6498.443,E2 -6498.443} C_VEL
LIN {X 0,Y 488.695,Z 277.232,A -85,B 0,C 180,E1 -6501.071,E2 -6501.071} C_VEL
LIN {X 0,Y 488.656,Z 277.239,A -85,B 0,C 180,E1 -6503.747,E2 -6503.747} C_VEL
LIN {X 0,Y 488.685,Z 277.235,A -85,B 0,C 180,E1 -6506.922,E2 -6506.922} C_VEL
LIN {X 0,Y 488.711,Z 277.237,A -85,B 0,C 180,E1 -6510.22,E2 -6510.22} C_VEL
LIN {X 0,Y 488.699,Z 277.229,A -85,B 0,C 180,E1 -6513.48,E2 -6513.48} C_VEL
LIN {X 0,Y 488.638,Z 277.243,A -85,B 0,C 180,E1 -6516.35,E2 -6516.35} C_VEL
LIN {X 0,Y 488.677,Z 277.232,A -85,B 0,C 180,E1 -6519.256,E2 -6519.256} C_VEL
LIN {X 0,Y 488.658,Z 277.24,A -85,B 0,C 180,E1 -6522.529,E2 -6522.529} C_VEL
LIN {X 0,Y 488.693,Z 277.233,A -85,B 0,C 180,E1 -6525.198,E2 -6525.198} C_VEL
LIN {X 0,Y 488.655,Z 277.239,A -85,B 0,C 180,E1 -6528.58,E2 -6528.58} C_VEL
LIN {X 0,Y 488.682,Z 277.234,A -85,B 0,C 180,E1 -6530.95,E2 -6530.95} C_VEL
LIN {X 0,Y 488.66,Z 277.243,A -85,B 0,C 180,E1 -6533.868,E2 -6533.868} C_VEL
LIN {X 0,Y 488.734,Z 277.23,A -85,B 0,C 180,E1 -6536.878,E2 -6536.878} C_VEL
LIN {X 0,Y 488.73,Z 277.234,A -85,B 0,C 180,E1 -6540.495,E2 -6540.495} C_VEL
LIN {X 0,Y 488.791,Z 277.636,A -85,B 0,C 180,E1 -6540.617,E2 -6540.617} C_VEL
LIN {X 0,Y 492.39,Z 292.709,A -85,B 0,C 180,E1 -6543.053,E2 -6543.053} C_VEL
LIN {X 0,Y 492.598,Z 297.443,A -85,B 0,C 180,E1 -6543.751,E2 -6543.751} C_VEL
LIN {X 0,Y 491.662,Z 317.85,A -85,B 0,C 180,E1 -6546.631,E2 -6546.631} C_VEL
LIN {X 0,Y 491.535,Z 319.928,A -85,B 0,C 180,E1 -6546.921,E2 -6546.921} C_VEL
LIN {X 0,Y 495.555,Z 341.315,A -85,B 0,C 180,E1 -6547.451,E2 -6547.451} C_VEL
LIN {X 0,Y 494.093,Z 486.921,A -85,B 0,C 180,E1 -6549.633,E2 -6549.633} C_VEL
LIN {X 0,Y 493.692,Z 502.561,A -85,B 0,C 180,E1 -6550.042,E2 -6550.042} C_VEL
LIN {X 0,Y 493.124,Z 517.171,A -85,B 0,C 180,E1 -6550.586,E2 -6550.586} C_VEL
LIN {X 0,Y 492.486,Z 531.164,A -85,B 0,C 180,E1 -6551.272,E2 -6551.272} C_VEL
LIN {X 0,Y 491.824,Z 544.678,A -85,B 0,C 180,E1 -6552.108,E2 -6552.108} C_VEL
LIN {X 0,Y 491.107,Z 557.141,A -85,B 0,C 180,E1 -6553.048,E2 -6553.048} C_VEL
LIN {X 0,Y 490.419,Z 569.82,A -85,B 0,C 180,E1 -6554.2,E2 -6554.2} C_VEL
LIN {X 0,Y 489.757,Z 581.342,A -85,B 0,C 180,E1 -6555.456,E2 -6555.456} C_VEL
LIN {X 0,Y 489.248,Z 591.042,A -85,B 0,C 180,E1 -6556.713,E2 -6556.713} C_VEL
LIN {X 0,Y 488.776,Z 600.742,A -85,B 0,C 180,E1 -6558.206,E2 -6558.206} C_VEL
LIN {X 0,Y 488.473,Z 608.513,A -85,B 0,C 180,E1 -6559.639,E2 -6559.639} C_VEL
LIN {X 0,Y 488.168,Z 615.927,A -85,B 0,C 180,E1 -6561.306,E2 -6561.306} C_VEL
LIN {X 0,Y 488.066,Z 621.811,A -85,B 0,C 180,E1 -6562.97,E2 -6562.97} C_VEL
LIN {X 0,Y 487.968,Z 625.307,A -85,B 0,C 180,E1 -6564.214,E2 -6564.214} C_VEL
LIN {X 0,Y 487.889,Z 628.84,A -85,B 0,C 180,E1 -6565.87,E2 -6565.87} C_VEL
LIN {X 0,Y 487.904,Z 631.166,A -85,B 0,C 180,E1 -6567.523,E2 -6567.523} C_VEL
LIN {X 0,Y 487.831,Z 632.335,A -85,B 0,C 180,E1 -6569.175,E2 -6569.175} C_VEL
LIN {X 0,Y 487.831,Z 632.334,A -85,B 0,C 180,E1 -6570.825,E2 -6570.825} C_VEL
LIN {X 0,Y 487.904,Z 631.162,A -85,B 0,C 180,E1 -6572.477,E2 -6572.477} C_VEL
LIN {X 0,Y 487.889,Z 628.836,A -85,B 0,C 180,E1 -6574.13,E2 -6574.13} C_VEL
LIN {X 0,Y 487.966,Z 625.308,A -85,B 0,C 180,E1 -6575.786,E2 -6575.786} C_VEL
LIN {X 0,Y 488.063,Z 620.487,A -85,B 0,C 180,E1 -6577.446,E2 -6577.446} C_VEL
LIN {X 0,Y 488.228,Z 614.243,A -85,B 0,C 180,E1 -6579.111,E2 -6579.111} C_VEL
LIN {X 0,Y 488.586,Z 606.405,A -85,B 0,C 180,E1 -6580.777,E2 -6580.777} C_VEL
LIN {X 0,Y 488.838,Z 598.687,A -85,B 0,C 180,E1 -6582.141,E2 -6582.141} C_VEL
LIN {X 0,Y 489.428,Z 588.028,A -85,B 0,C 180,E1 -6583.705,E2 -6583.705} C_VEL
LIN {X 0,Y 489.947,Z 577.758,A -85,B 0,C 180,E1 -6584.963,E2 -6584.963} C_VEL
LIN {X 0,Y 490.622,Z 566.038,A -85,B 0,C 180,E1 -6586.169,E2 -6586.169} C_VEL
LIN {X 0,Y 491.316,Z 553.258,A -85,B 0,C 180,E1 -6587.266,E2 -6587.266} C_VEL
LIN {X 0,Y 492.116,Z 539.912,A -85,B 0,C 180,E1 -6588.203,E2 -6588.203} C_VEL
LIN {X 0,Y 492.7,Z 527.173,A -85,B 0,C 180,E1 -6588.935,E2 -6588.935} C_VEL
LIN {X 0,Y 493.305,Z 512.662,A -85,B 0,C 180,E1 -6589.596,E2 -6589.596} C_VEL
LIN {X 0,Y 493.778,Z 497.134,A -85,B 0,C 180,E1 -6590.12,E2 -6590.12} C_VEL
LIN {X 0,Y 494.161,Z 482.564,A -85,B 0,C 180,E1 -6590.445,E2 -6590.445} C_VEL
LIN {X 0,Y 495.552,Z 340.344,A -85,B 0,C 180,E1 -6592.563,E2 -6592.563} C_VEL
LIN {X 0,Y 491.541,Z 319.926,A -85,B 0,C 180,E1 -6593.077,E2 -6593.077} C_VEL
LIN {X 0,Y 492.543,Z 299.301,A -85,B 0,C 180,E1 -6595.982,E2 -6595.982} C_VEL
LIN {X 0,Y 492.644,Z 294.283,A -85,B 0,C 180,E1 -6596.703,E2 -6596.703} C_VEL
LIN {X 0,Y 489.26,Z 279.545,A -85,B 0,C 180,E1 -6599.066,E2 -6599.066} C_VEL
LIN {X 0,Y 488.723,Z 277.234,A -85,B 0,C 180,E1 -6599.447,E2 -6599.447} C_VEL
LIN {X 0,Y 488.699,Z 277.232,A -85,B 0,C 180,E1 -6602.146,E2 -6602.146} C_VEL
LIN {X 0,Y 488.709,Z 277.231,A -85,B 0,C 180,E1 -6605.115,E2 -6605.115} C_VEL
LIN {X 0,Y 488.652,Z 277.244,A -85,B 0,C 180,E1 -6608.201,E2 -6608.201} C_VEL
LIN {X 0,Y 488.686,Z 277.239,A -85,B 0,C 180,E1 -6610.34,E2 -6610.34} C_VEL
LIN {X 0,Y 488.665,Z 277.241,A -85,B 0,C 180,E1 -6613.655,E2 -6613.655} C_VEL
LIN {X 0,Y 488.666,Z 277.24,A -85,B 0,C 180,E1 -6616.343,E2 -6616.343} C_VEL
LIN {X 0,Y 488.694,Z 277.237,A -85,B 0,C 180,E1 -6619.673,E2 -6619.673} C_VEL
LIN {X 0,Y 488.64,Z 277.239,A -85,B 0,C 180,E1 -6622.838,E2 -6622.838} C_VEL
LIN {X 0,Y 488.707,Z 277.237,A -85,B 0,C 180,E1 -6625.885,E2 -6625.885} C_VEL
LIN {X 0,Y 488.679,Z 277.234,A -85,B 0,C 180,E1 -6628.819,E2 -6628.819} C_VEL
LIN {X 0,Y 488.696,Z 277.239,A -85,B 0,C 180,E1 -6631.668,E2 -6631.668} C_VEL
LIN {X 0,Y 488.684,Z 277.234,A -85,B 0,C 180,E1 -6634.959,E2 -6634.959} C_VEL
LIN {X 0,Y 488.685,Z 277.236,A -85,B 0,C 180,E1 -6638.043,E2 -6638.043} C_VEL
LIN {X 0,Y 488.721,Z 277.219,A -85,B 0,C 180,E1 -6640.686,E2 -6640.686} C_VEL
LIN {X 0,Y 488.744,Z 277.228,A -85,B 0,C 180,E1 -6644.144,E2 -6644.144} C_VEL
LIN {X 0,Y 488.723,Z 277.223,A -85,B 0,C 180,E1 -6647.543,E2 -6647.543} C_VEL
LIN {X 0,Y 488.711,Z 277.228,A -85,B 0,C 180,E1 -6650.063,E2 -6650.063} C_VEL
LIN {X 0,Y 488.832,Z 277.215,A -85,B 0,C 180,E1 -6652.744,E2 -6652.744} C_VEL
LIN {X 0,Y 488.784,Z 277.22,A -85,B 0,C 180,E1 -6655.051,E2 -6655.051} C_VEL
LIN {X 0,Y 488.931,Z 277.206,A -85,B 0,C 180,E1 -6657.529,E2 -6657.529} C_VEL
LIN {X 0,Y 488.924,Z 277.205,A -85,B 0,C 180,E1 -6660,E2 -6660} C_VEL
LIN {X 0,Y 488.935,Z 277.199,A -85,B 0,C 180,E1 -6662.472,E2 -6662.472} C_VEL
LIN {X 0,Y 488.821,Z 277.217,A -85,B 0,C 180,E1 -6665.776,E2 -6665.776} C_VEL
LIN {X 0,Y 488.769,Z 277.222,A -85,B 0,C 180,E1 -6668.267,E2 -6668.267} C_VEL
LIN {X 0,Y 488.791,Z 277.223,A -85,B 0,C 180,E1 -6671.613,E2 -6671.613} C_VEL
LIN {X 0,Y 488.74,Z 277.23,A -85,B 0,C 180,E1 -6675.001,E2 -6675.001} C_VEL
LIN {X 0,Y 488.733,Z 277.227,A -85,B 0,C 180,E1 -6678.443,E2 -6678.443} C_VEL
LIN {X 0,Y 488.695,Z 277.227,A -85,B 0,C 180,E1 -6681.071,E2 -6681.071} C_VEL
LIN {X 0,Y 488.659,Z 277.237,A -85,B 0,C 180,E1 -6683.747,E2 -6683.747} C_VEL
LIN {X 0,Y 488.737,Z 277.224,A -85,B 0,C 180,E1 -6686.934,E2 -6686.934} C_VEL
LIN {X 0,Y 488.711,Z 277.234,A -85,B 0,C 180,E1 -6689.271,E2 -6689.271} C_VEL
LIN {X 0,Y 488.687,Z 277.231,A -85,B 0,C 180,E1 -6692.148,E2 -6692.148} C_VEL
LIN {X 0,Y 488.706,Z 277.236,A -85,B 0,C 180,E1 -6695.116,E2 -6695.116} C_VEL
LIN {X 0,Y 488.671,Z 277.234,A -85,B 0,C 180,E1 -6698.201,E2 -6698.201} C_VEL
LIN {X 0,Y 488.711,Z 277.231,A -85,B 0,C 180,E1 -6700.346,E2 -6700.346} C_VEL
LIN {X 0,Y 488.677,Z 277.235,A -85,B 0,C 180,E1 -6703.656,E2 -6703.656} C_VEL
LIN {X 0,Y 488.678,Z 277.238,A -85,B 0,C 180,E1 -6706.346,E2 -6706.346} C_VEL
LIN {X 0,Y 488.728,Z 277.229,A -85,B 0,C 180,E1 -6709.677,E2 -6709.677} C_VEL
LIN {X 0,Y 488.675,Z 277.24,A -85,B 0,C 180,E1 -6712.842,E2 -6712.842} C_VEL
LIN {X 0,Y 488.721,Z 277.231,A -85,B 0,C 180,E1 -6715.888,E2 -6715.888} C_VEL
LIN {X 0,Y 488.689,Z 277.237,A -85,B 0,C 180,E1 -6718.821,E2 -6718.821} C_VEL
LIN {X 0,Y 488.741,Z 277.23,A -85,B 0,C 180,E1 -6721.672,E2 -6721.672} C_VEL
LIN {X 0,Y 488.79,Z 277.216,A -85,B 0,C 180,E1 -6723.061,E2 -6723.061} C_VEL
LIN {X 0,Y 488.561,Z 277.735,A -85,B 0,C 180,E1 -6723.513,E2 -6723.513} C_VEL
LIN {X 0,Y 488.061,Z 279.052,A -85,B 0,C 180,E1 -6723.943,E2 -6723.943} C_VEL
LIN {X 0,Y 486.658,Z 283.1,A -85,B 0,C 180,E1 -6724.736,E2 -6724.736} C_VEL
LIN {X 0,Y 484.904,Z 290.423,A -85,B 0,C 180,E1 -6725.87,E2 -6725.87} C_VEL
LIN {X 0,Y 484.821,Z 292.75,A -85,B 0,C 180,E1 -6726.258,E2 -6726.258} C_VEL
LIN {X 0,Y 484.849,Z 295.052,A -85,B 0,C 180,E1 -6726.642,E2 -6726.642} C_VEL
LIN {X 0,Y 489.063,Z 313.094,A -85,B 0,C 180,E1 -6727.146,E2 -6727.146} C_VEL
LIN {X 0,Y 488.037,Z 421.874,A -85,B 0,C 180,E1 -6728.789,E2 -6728.789} C_VEL
LIN {X 0,Y 487.612,Z 460.441,A -85,B 0,C 180,E1 -6729.391,E2 -6729.391} C_VEL
LIN {X 0,Y 487.225,Z 475.709,A -85,B 0,C 180,E1 -6729.792,E2 -6729.792} C_VEL
LIN {X 0,Y 486.733,Z 490.415,A -85,B 0,C 180,E1 -6730.349,E2 -6730.349} C_VEL
LIN {X 0,Y 486.054,Z 503.862,A -85,B 0,C 180,E1 -6731.015,E2 -6731.015} C_VEL
LIN {X 0,Y 485.385,Z 517.452,A -85,B 0,C 180,E1 -6731.863,E2 -6731.863} C_VEL
LIN {X 0,Y 484.65,Z 529.946,A -85,B 0,C 180,E1 -6732.815,E2 -6732.815} C_VEL
LIN {X 0,Y 483.849,Z 542.595,A -85,B 0,C 180,E1 -6733.98,E2 -6733.98} C_VEL
LIN {X 0,Y 483.154,Z 554.058,A -85,B 0,C 180,E1 -6735.253,E2 -6735.253} C_VEL
LIN {X 0,Y 482.595,Z 563.702,A -85,B 0,C 180,E1 -6736.526,E2 -6736.526} C_VEL
LIN {X 0,Y 482.026,Z 573.19,A -85,B 0,C 180,E1 -6738.015,E2 -6738.015} C_VEL
LIN {X 0,Y 481.619,Z 581.019,A -85,B 0,C 180,E1 -6739.49,E2 -6739.49} C_VEL
LIN {X 0,Y 481.292,Z 588.361,A -85,B 0,C 180,E1 -6741.181,E2 -6741.181} C_VEL
LIN {X 0,Y 481.077,Z 594.187,A -85,B 0,C 180,E1 -6742.867,E2 -6742.867} C_VEL
LIN {X 0,Y 481.016,Z 597.634,A -85,B 0,C 180,E1 -6744.13,E2 -6744.13} C_VEL
LIN {X 0,Y 480.865,Z 601.134,A -85,B 0,C 180,E1 -6745.809,E2 -6745.809} C_VEL
LIN {X 0,Y 480.841,Z 603.449,A -85,B 0,C 180,E1 -6747.487,E2 -6747.487} C_VEL
LIN {X 0,Y 480.757,Z 604.635,A -85,B 0,C 180,E1 -6749.162,E2 -6749.162} C_VEL
LIN {X 0,Y 480.757,Z 604.653,A -85,B 0,C 180,E1 -6750.838,E2 -6750.838} C_VEL
LIN {X 0,Y 480.842,Z 603.538,A -85,B 0,C 180,E1 -6752.513,E2 -6752.513} C_VEL
LIN {X 0,Y 480.864,Z 601.293,A -85,B 0,C 180,E1 -6754.191,E2 -6754.191} C_VEL
LIN {X 0,Y 481.009,Z 597.859,A -85,B 0,C 180,E1 -6755.87,E2 -6755.87} C_VEL
LIN {X 0,Y 481.133,Z 593.161,A -85,B 0,C 180,E1 -6757.554,E2 -6757.554} C_VEL
LIN {X 0,Y 481.342,Z 587.071,A -85,B 0,C 180,E1 -6759.242,E2 -6759.242} C_VEL
LIN {X 0,Y 481.764,Z 579.399,A -85,B 0,C 180,E1 -6760.932,E2 -6760.932} C_VEL
LIN {X 0,Y 482.127,Z 571.305,A -85,B 0,C 180,E1 -6762.402,E2 -6762.402} C_VEL
LIN {X 0,Y 482.739,Z 561.364,A -85,B 0,C 180,E1 -6763.899,E2 -6763.899} C_VEL
LIN {X 0,Y 483.366,Z 551.256,A -85,B 0,C 180,E1 -6765.171,E2 -6765.171} C_VEL
LIN {X 0,Y 484.032,Z 540.79,A -85,B 0,C 180,E1 -6766.287,E2 -6766.287} C_VEL
LIN {X 0,Y 484.738,Z 528.438,A -85,B 0,C 180,E1 -6767.399,E2 -6767.399} C_VEL
LIN {X 0,Y 485.543,Z 515.611,A -85,B 0,C 180,E1 -6768.349,E2 -6768.349} C_VEL
LIN {X 0,Y 486.213,Z 501.545,A -85,B 0,C 180,E1 -6769.198,E2 -6769.198} C_VEL
LIN {X 0,Y 486.863,Z 487.126,A -85,B 0,C 180,E1 -6769.876,E2 -6769.876} C_VEL
LIN {X 0,Y 487.287,Z 472.134,A -85,B 0,C 180,E1 -6770.405,E2 -6770.405} C_VEL
LIN {X 0,Y 487.614,Z 457.543,A -85,B 0,C 180,E1 -6770.755,E2 -6770.755} C_VEL
LIN {X 0,Y 488.427,Z 378.607,A -85,B 0,C 180,E1 -6771.955,E2 -6771.955} C_VEL
LIN {X 0,Y 488.982,Z 313.031,A -85,B 0,C 180,E1 -6772.951,E2 -6772.951} C_VEL
LIN {X 0,Y 484.889,Z 295.038,A -85,B 0,C 180,E1 -6773.448,E2 -6773.448} C_VEL
LIN {X 0,Y 484.555,Z 290.873,A -85,B 0,C 180,E1 -6774.165,E2 -6774.165} C_VEL
LIN {X 0,Y 481.718,Z 278.106,A -85,B 0,C 180,E1 -6776.538,E2 -6776.538} C_VEL
LIN {X 0,Y 481.676,Z 278.114,A -85,B 0,C 180,E1 -6779.74,E2 -6779.74} C_VEL
LIN {X 0,Y 481.669,Z 278.111,A -85,B 0,C 180,E1 -6782.673,E2 -6782.673} C_VEL
LIN {X 0,Y 481.638,Z 278.12,A -85,B 0,C 180,E1 -6785.708,E2 -6785.708} C_VEL
LIN {X 0,Y 481.667,Z 278.113,A -85,B 0,C 180,E1 -6788.858,E2 -6788.858} C_VEL
LIN {X 0,Y 481.647,Z 278.113,A -85,B 0,C 180,E1 -6791.912,E2 -6791.912} C_VEL
LIN {X 0,Y 481.649,Z 278.111,A -85,B 0,C 180,E1 -6794.457,E2 -6794.457} C_VEL
LIN {X 0,Y 481.638,Z 278.105,A -85,B 0,C 180,E1 -6797.838,E2 -6797.838} C_VEL
LIN {X 0,Y 481.652,Z 278.111,A -85,B 0,C 180,E1 -6800.653,E2 -6800.653} C_VEL
LIN {X 0,Y 481.619,Z 278.111,A -85,B 0,C 180,E1 -6803.375,E2 -6803.375} C_VEL
LIN {X 0,Y 481.661,Z 278.109,A -85,B 0,C 180,E1 -6806.326,E2 -6806.326} C_VEL
LIN {X 0,Y 481.639,Z 278.105,A -85,B 0,C 180,E1 -6809.417,E2 -6809.417} C_VEL
LIN {X 0,Y 481.681,Z 278.105,A -85,B 0,C 180,E1 -6812.167,E2 -6812.167} C_VEL
LIN {X 0,Y 481.667,Z 278.111,A -85,B 0,C 180,E1 -6814.967,E2 -6814.967} C_VEL
LIN {X 0,Y 481.636,Z 278.109,A -85,B 0,C 180,E1 -6817.704,E2 -6817.704} C_VEL
LIN {X 0,Y 481.69,Z 278.106,A -85,B 0,C 180,E1 -6820.392,E2 -6820.392} C_VEL
LIN {X 0,Y 481.663,Z 278.113,A -85,B 0,C 180,E1 -6823.033,E2 -6823.033} C_VEL
LIN {X 0,Y 481.67,Z 278.106,A -85,B 0,C 180,E1 -6825.638,E2 -6825.638} C_VEL
LIN {X 0,Y 481.737,Z 278.099,A -85,B 0,C 180,E1 -6828.215,E2 -6828.215} C_VEL
LIN {X 0,Y 481.724,Z 278.098,A -85,B 0,C 180,E1 -6831.611,E2 -6831.611} C_VEL
LIN {X 0,Y 481.783,Z 278.094,A -85,B 0,C 180,E1 -6834.139,E2 -6834.139} C_VEL
LIN {X 0,Y 481.903,Z 278.079,A -85,B 0,C 180,E1 -6837.492,E2 -6837.492} C_VEL
LIN {X 0,Y 481.921,Z 278.074,A -85,B 0,C 180,E1 -6840,E2 -6840} C_VEL
LIN {X 0,Y 481.899,Z 278.085,A -85,B 0,C 180,E1 -6842.508,E2 -6842.508} C_VEL
LIN {X 0,Y 481.781,Z 278.092,A -85,B 0,C 180,E1 -6845.861,E2 -6845.861} C_VEL
LIN {X 0,Y 481.713,Z 278.108,A -85,B 0,C 180,E1 -6848.389,E2 -6848.389} C_VEL
LIN {X 0,Y 481.736,Z 278.1,A -85,B 0,C 180,E1 -6851.785,E2 -6851.785} C_VEL
LIN {X 0,Y 481.728,Z 278.101,A -85,B 0,C 180,E1 -6855.225,E2 -6855.225} C_VEL
LIN {X 0,Y 481.693,Z 278.109,A -85,B 0,C 180,E1 -6858.722,E2 -6858.722} C_VEL
LIN {X 0,Y 481.633,Z 278.111,A -85,B 0,C 180,E1 -6861.395,E2 -6861.395} C_VEL
LIN {X 0,Y 481.635,Z 278.118,A -85,B 0,C 180,E1 -6864.115,E2 -6864.115} C_VEL
LIN {X 0,Y 481.66,Z 278.109,A -85,B 0,C 180,E1 -6867.122,E2 -6867.122} C_VEL
LIN {X 0,Y 481.66,Z 278.111,A -85,B 0,C 180,E1 -6869.742,E2 -6869.742} C_VEL
LIN {X 0,Y 481.641,Z 278.11,A -85,B 0,C 180,E1 -6872.676,E2 -6872.676} C_VEL
LIN {X 0,Y 481.638,Z 278.111,A -85,B 0,C 180,E1 -6875.202,E2 -6875.202} C_VEL
LIN {X 0,Y 481.62,Z 278.12,A -85,B 0,C 180,E1 -6878.004,E2 -6878.004} C_VEL
LIN {X 0,Y 481.622,Z 278.106,A -85,B 0,C 180,E1 -6881.045,E2 -6881.045} C_VEL
LIN {X 0,Y 481.646,Z 278.114,A -85,B 0,C 180,E1 -6884.459,E2 -6884.459} C_VEL
LIN {X 0,Y 481.608,Z 278.116,A -85,B 0,C 180,E1 -6886.856,E2 -6886.856} C_VEL
LIN {X 0,Y 481.649,Z 278.115,A -85,B 0,C 180,E1 -6890.058,E2 -6890.058} C_VEL
LIN {X 0,Y 481.612,Z 278.116,A -85,B 0,C 180,E1 -6893.379,E2 -6893.379} C_VEL
LIN {X 0,Y 481.689,Z 278.11,A -85,B 0,C 180,E1 -6896.329,E2 -6896.329} C_VEL
LIN {X 0,Y 481.688,Z 278.112,A -85,B 0,C 180,E1 -6899.778,E2 -6899.778} C_VEL
LIN {X 0,Y 481.708,Z 278.228,A -85,B 0,C 180,E1 -6900.262,E2 -6900.262} C_VEL
LIN {X 0,Y 485.489,Z 294.089,A -85,B 0,C 180,E1 -6902.872,E2 -6902.872} C_VEL
LIN {X 0,Y 485.862,Z 297.252,A -85,B 0,C 180,E1 -6903.359,E2 -6903.359} C_VEL
LIN {X 0,Y 484.752,Z 319.699,A -85,B 0,C 180,E1 -6906.576,E2 -6906.576} C_VEL
LIN {X 0,Y 489.013,Z 341.97,A -85,B 0,C 180,E1 -6907.146,E2 -6907.146} C_VEL
LIN {X 0,Y 487.443,Z 486.726,A -85,B 0,C 180,E1 -6909.343,E2 -6909.343} C_VEL
LIN {X 0,Y 486.974,Z 502.51,A -85,B 0,C 180,E1 -6909.76,E2 -6909.76} C_VEL
LIN {X 0,Y 486.397,Z 517.226,A -85,B 0,C 180,E1 -6910.318,E2 -6910.318} C_VEL
LIN {X 0,Y 485.741,Z 530.964,A -85,B 0,C 180,E1 -6911.002,E2 -6911.002} C_VEL
LIN {X 0,Y 485.044,Z 544.476,A -85,B 0,C 180,E1 -6911.85,E2 -6911.85} C_VEL
LIN {X 0,Y 484.255,Z 556.937,A -85,B 0,C 180,E1 -6912.801,E2 -6912.801} C_VEL
LIN {X 0,Y 483.599,Z 568.138,A -85,B 0,C 180,E1 -6913.823,E2 -6913.823} C_VEL
LIN {X 0,Y 482.877,Z 579.344,A -85,B 0,C 180,E1 -6915.029,E2 -6915.029} C_VEL
LIN {X 0,Y 482.358,Z 589.343,A -85,B 0,C 180,E1 -6916.305,E2 -6916.305} C_VEL
LIN {X 0,Y 481.777,Z 599.121,A -85,B 0,C 180,E1 -6917.788,E2 -6917.788} C_VEL
LIN {X 0,Y 481.49,Z 607.294,A -85,B 0,C 180,E1 -6919.275,E2 -6919.275} C_VEL
LIN {X 0,Y 481.175,Z 614.042,A -85,B 0,C 180,E1 -6920.755,E2 -6920.755} C_VEL
LIN {X 0,Y 480.987,Z 620.279,A -85,B 0,C 180,E1 -6922.444,E2 -6922.444} C_VEL
LIN {X 0,Y 480.876,Z 625.103,A -85,B 0,C 180,E1 -6924.128,E2 -6924.128} C_VEL
LIN {X 0,Y 480.792,Z 628.637,A -85,B 0,C 180,E1 -6925.809,E2 -6925.809} C_VEL
LIN {X 0,Y 480.818,Z 630.963,A -85,B 0,C 180,E1 -6927.487,E2 -6927.487} C_VEL
LIN {X 0,Y 480.757,Z 632.132,A -85,B 0,C 180,E1 -6929.162,E2 -6929.162} C_VEL
LIN {X 0,Y 480.757,Z 632.132,A -85,B 0,C 180,E1 -6930.838,E2 -6930.838} C_VEL
LIN {X 0,Y 480.818,Z 630.959,A -85,B 0,C 180,E1 -6932.513,E2 -6932.513} C_VEL
LIN {X 0,Y 480.792,Z 628.632,A -85,B 0,C 180,E1 -6934.191,E2 -6934.191} C_VEL
LIN {X 0,Y 480.872,Z 625.104,A -85,B 0,C 180,E1 -6935.872,E2 -6935.872} C_VEL
LIN {X 0,Y 480.987,Z 620.283,A -85,B 0,C 180,E1 -6937.556,E2 -6937.556} C_VEL
LIN {X 0,Y 481.175,Z 614.039,A -85,B 0,C 180,E1 -6939.245,E2 -6939.245} C_VEL
LIN {X 0,Y 481.565,Z 606.201,A -85,B 0,C 180,E1 -6940.936,E2 -6940.936} C_VEL
LIN {X 0,Y 481.856,Z 598.326,A -85,B 0,C 180,E1 -6942.347,E2 -6942.347} C_VEL
LIN {X 0,Y 482.452,Z 587.822,A -85,B 0,C 180,E1 -6943.907,E2 -6943.907} C_VEL
LIN {X 0,Y 483.016,Z 577.552,A -85,B 0,C 180,E1 -6945.183,E2 -6945.183} C_VEL
LIN {X 0,Y 483.702,Z 566.588,A -85,B 0,C 180,E1 -6946.331,E2 -6946.331} C_VEL
LIN {X 0,Y 484.395,Z 554.348,A -85,B 0,C 180,E1 -6947.412,E2 -6947.412} C_VEL
LIN {X 0,Y 485.21,Z 541.292,A -85,B 0,C 180,E1 -6948.362,E2 -6948.362} C_VEL
LIN {X 0,Y 485.968,Z 526.967,A -85,B 0,C 180,E1 -6949.208,E2 -6949.208} C_VEL
LIN {X 0,Y 486.578,Z 513.046,A -85,B 0,C 180,E1 -6949.854,E2 -6949.854} C_VEL
LIN {X 0,Y 487.088,Z 497.75,A -85,B 0,C 180,E1 -6950.383,E2 -6950.383} C_VEL
LIN {X 0,Y 487.508,Z 482.35,A -85,B 0,C 180,E1 -6950.737,E2 -6950.737} C_VEL
LIN {X 0,Y 488.984,Z 342.108,A -85,B 0,C 180,E1 -6952.853,E2 -6952.853} C_VEL
LIN {X 0,Y 484.761,Z 319.715,A -85,B 0,C 180,E1 -6953.42,E2 -6953.42} C_VEL
LIN {X 0,Y 485.82,Z 299.159,A -85,B 0,C 180,E1 -6956.361,E2 -6956.361} C_VEL
LIN {X 0,Y 485.76,Z 295.661,A -85,B 0,C 180,E1 -6956.879,E2 -6956.879} C_VEL
LIN {X 0,Y 482.609,Z 282.011,A -85,B 0,C 180,E1 -6959.103,E2 -6959.103} C_VEL
LIN {X 0,Y 481.68,Z 278.11,A -85,B 0,C 180,E1 -6959.77,E2 -6959.77} C_VEL
LIN {X 0,Y 481.667,Z 278.11,A -85,B 0,C 180,E1 -6962.673,E2 -6962.673} C_VEL
LIN {X 0,Y 481.624,Z 278.117,A -85,B 0,C 180,E1 -6965.709,E2 -6965.709} C_VEL
LIN {X 0,Y 481.626,Z 278.115,A -85,B 0,C 180,E1 -6968.862,E2 -6968.862} C_VEL
LIN {X 0,Y 481.617,Z 278.121,A -85,B 0,C 180,E1 -6971.908,E2 -6971.908} C_VEL
LIN {X 0,Y 481.646,Z 278.114,A -85,B 0,C 180,E1 -6974.457,E2 -6974.457} C_VEL
LIN {X 0,Y 481.62,Z 278.119,A -85,B 0,C 180,E1 -6977.836,E2 -6977.836} C_VEL
LIN {X 0,Y 481.639,Z 278.112,A -85,B 0,C 180,E1 -6980.655,E2 -6980.655} C_VEL
LIN {X 0,Y 481.598,Z 278.118,A -85,B 0,C 180,E1 -6983.379,E2 -6983.379} C_VEL
LIN {X 0,Y 481.66,Z 278.109,A -85,B 0,C 180,E1 -6986.326,E2 -6986.326} C_VEL
LIN {X 0,Y 481.637,Z 278.114,A -85,B 0,C 180,E1 -6989.417,E2 -6989.417} C_VEL
LIN {X 0,Y 481.646,Z 278.111,A -85,B 0,C 180,E1 -6992.165,E2 -6992.165} C_VEL
LIN {X 0,Y 481.658,Z 278.109,A -85,B 0,C 180,E1 -6994.967,E2 -6994.967} C_VEL
LIN {X 0,Y 481.636,Z 278.119,A -85,B 0,C 180,E1 -6997.704,E2 -6997.704} C_VEL
LIN {X 0,Y 481.687,Z 278.096,A -85,B 0,C 180,E1 -7000.392,E2 -7000.392} C_VEL
LIN {X 0,Y 481.651,Z 278.107,A -85,B 0,C 180,E1 -7003.033,E2 -7003.033} C_VEL
LIN {X 0,Y 481.662,Z 278.112,A -85,B 0,C 180,E1 -7005.638,E2 -7005.638} C_VEL
LIN {X 0,Y 481.719,Z 278.086,A -85,B 0,C 180,E1 -7008.214,E2 -7008.214} C_VEL
LIN {X 0,Y 481.701,Z 278.11,A -85,B 0,C 180,E1 -7011.611,E2 -7011.611} C_VEL
LIN {X 0,Y 481.78,Z 278.09,A -85,B 0,C 180,E1 -7014.139,E2 -7014.139} C_VEL
LIN {X 0,Y 481.898,Z 278.083,A -85,B 0,C 180,E1 -7017.492,E2 -7017.492} C_VEL
LIN {X 0,Y 481.893,Z 278.081,A -85,B 0,C 180,E1 -7020,E2 -7020} C_VEL
LIN {X 0,Y 481.902,Z 278.076,A -85,B 0,C 180,E1 -7022.508,E2 -7022.508} C_VEL
LIN {X 0,Y 481.782,Z 278.093,A -85,B 0,C 180,E1 -7025.861,E2 -7025.861} C_VEL
LIN {X 0,Y 481.724,Z 278.1,A -85,B 0,C 180,E1 -7028.389,E2 -7028.389} C_VEL
LIN {X 0,Y 481.737,Z 278.1,A -85,B 0,C 180,E1 -7031.785,E2 -7031.785} C_VEL
LIN {X 0,Y 481.725,Z 278.105,A -85,B 0,C 180,E1 -7035.225,E2 -7035.225} C_VEL
LIN {X 0,Y 481.695,Z 278.106,A -85,B 0,C 180,E1 -7038.722,E2 -7038.722} C_VEL
LIN {X 0,Y 481.633,Z 278.109,A -85,B 0,C 180,E1 -7041.395,E2 -7041.395} C_VEL
LIN {X 0,Y 481.638,Z 278.111,A -85,B 0,C 180,E1 -7044.115,E2 -7044.115} C_VEL
LIN {X 0,Y 481.704,Z 278.098,A -85,B 0,C 180,E1 -7047.132,E2 -7047.132} C_VEL
LIN {X 0,Y 481.667,Z 278.108,A -85,B 0,C 180,E1 -7049.742,E2 -7049.742} C_VEL
LIN {X 0,Y 481.643,Z 278.113,A -85,B 0,C 180,E1 -7052.677,E2 -7052.677} C_VEL
LIN {X 0,Y 481.627,Z 278.112,A -85,B 0,C 180,E1 -7055.71,E2 -7055.71} C_VEL
LIN {X 0,Y 481.662,Z 278.115,A -85,B 0,C 180,E1 -7058.86,E2 -7058.86} C_VEL
LIN {X 0,Y 481.645,Z 278.11,A -85,B 0,C 180,E1 -7061.914,E2 -7061.914} C_VEL
LIN {X 0,Y 481.648,Z 278.114,A -85,B 0,C 180,E1 -7064.459,E2 -7064.459} C_VEL
LIN {X 0,Y 481.642,Z 278.112,A -85,B 0,C 180,E1 -7067.84,E2 -7067.84} C_VEL
LIN {X 0,Y 481.675,Z 278.11,A -85,B 0,C 180,E1 -7070.652,E2 -7070.652} C_VEL
LIN {X 0,Y 481.623,Z 278.113,A -85,B 0,C 180,E1 -7073.377,E2 -7073.377} C_VEL
LIN {X 0,Y 481.674,Z 278.112,A -85,B 0,C 180,E1 -7076.328,E2 -7076.328} C_VEL
LIN {X 0,Y 481.648,Z 278.113,A -85,B 0,C 180,E1 -7079.418,E2 -7079.418} C_VEL
LIN {X 0,Y 481.697,Z 278.107,A -85,B 0,C 180,E1 -7082.169,E2 -7082.169} C_VEL
LIN {X 0,Y 481.723,Z 278.151,A -85,B 0,C 180,E1 -7083.579,E2 -7083.579} C_VEL
LIN {X 0,Y 484.64,Z 291.531,A -85,B 0,C 180,E1 -7086.044,E2 -7086.044} C_VEL
LIN {X 0,Y 484.821,Z 292.75,A -85,B 0,C 180,E1 -7086.258,E2 -7086.258} C_VEL
LIN {X 0,Y 485.476,Z 294.934,A -85,B 0,C 180,E1 -7086.54,E2 -7086.54} C_VEL
LIN {X 0,Y 487.371,Z 298.929,A -85,B 0,C 180,E1 -7086.823,E2 -7086.823} C_VEL
LIN {X 0,Y 488.395,Z 302.815,A -85,B 0,C 180,E1 -7086.951,E2 -7086.951} C_VEL
LIN {X 0,Y 487.946,Z 306.257,A -85,B 0,C 180,E1 -7086.982,E2 -7086.982} C_VEL
LIN {X 0,Y 484.109,Z 315.403,A -85,B 0,C 180,E1 -7086.932,E2 -7086.932} C_VEL
LIN {X 0,Y 482.526,Z 323.889,A -85,B 0,C 180,E1 -7086.986,E2 -7086.986} C_VEL
LIN {X 0,Y 480.981,Z 460.664,A -85,B 0,C 180,E1 -7089.094,E2 -7089.094} C_VEL
LIN {X 0,Y 480.557,Z 475.926,A -85,B 0,C 180,E1 -7089.499,E2 -7089.499} C_VEL
LIN {X 0,Y 480.051,Z 490.841,A -85,B 0,C 180,E1 -7090.074,E2 -7090.074} C_VEL
LIN {X 0,Y 479.355,Z 504.073,A -85,B 0,C 180,E1 -7090.739,E2 -7090.739} C_VEL
LIN {X 0,Y 478.629,Z 517.662,A -85,B 0,C 180,E1 -7091.598,E2 -7091.598} C_VEL
LIN {X 0,Y 477.844,Z 530.156,A -85,B 0,C 180,E1 -7092.563,E2 -7092.563} C_VEL
LIN {X 0,Y 477.024,Z 542.803,A -85,B 0,C 180,E1 -7093.745,E2 -7093.745} C_VEL
LIN {X 0,Y 476.274,Z 554.266,A -85,B 0,C 180,E1 -7095.035,E2 -7095.035} C_VEL
LIN {X 0,Y 475.647,Z 563.91,A -85,B 0,C 180,E1 -7096.326,E2 -7096.326} C_VEL
LIN {X 0,Y 475.026,Z 572.668,A -85,B 0,C 180,E1 -7097.706,E2 -7097.706} C_VEL
LIN {X 0,Y 474.681,Z 580.223,A -85,B 0,C 180,E1 -7099.119,E2 -7099.119} C_VEL
LIN {X 0,Y 474.32,Z 586.892,A -85,B 0,C 180,E1 -7100.62,E2 -7100.62} C_VEL
LIN {X 0,Y 474.062,Z 593.069,A -85,B 0,C 180,E1 -7102.333,E2 -7102.333} C_VEL
LIN {X 0,Y 473.94,Z 597.839,A -85,B 0,C 180,E1 -7104.042,E2 -7104.042} C_VEL
LIN {X 0,Y 473.771,Z 601.339,A -85,B 0,C 180,E1 -7105.747,E2 -7105.747} C_VEL
LIN {X 0,Y 473.758,Z 603.652,A -85,B 0,C 180,E1 -7107.449,E2 -7107.449} C_VEL
LIN {X 0,Y 473.686,Z 604.838,A -85,B 0,C 180,E1 -7109.15,E2 -7109.15} C_VEL
LIN {X 0,Y 473.686,Z 604.855,A -85,B 0,C 180,E1 -7110.85,E2 -7110.85} C_VEL
LIN {X 0,Y 473.758,Z 603.74,A -85,B 0,C 180,E1 -7112.551,E2 -7112.551} C_VEL
LIN {X 0,Y 473.77,Z 601.495,A -85,B 0,C 180,E1 -7114.253,E2 -7114.253} C_VEL
LIN {X 0,Y 473.933,Z 598.061,A -85,B 0,C 180,E1 -7115.958,E2 -7115.958} C_VEL
LIN {X 0,Y 474.062,Z 593.363,A -85,B 0,C 180,E1 -7117.667,E2 -7117.667} C_VEL
LIN {X 0,Y 474.293,Z 587.273,A -85,B 0,C 180,E1 -7119.381,E2 -7119.381} C_VEL
LIN {X 0,Y 474.78,Z 579.6,A -85,B 0,C 180,E1 -7121.095,E2 -7121.095} C_VEL
LIN {X 0,Y 475.137,Z 571.918,A -85,B 0,C 180,E1 -7122.514,E2 -7122.514} C_VEL
LIN {X 0,Y 475.816,Z 561.565,A -85,B 0,C 180,E1 -7124.105,E2 -7124.105} C_VEL
LIN {X 0,Y 476.472,Z 551.456,A -85,B 0,C 180,E1 -7125.396,E2 -7125.396} C_VEL
LIN {X 0,Y 477.175,Z 541.293,A -85,B 0,C 180,E1 -7126.496,E2 -7126.496} C_VEL
LIN {X 0,Y 477.936,Z 528.636,A -85,B 0,C 180,E1 -7127.655,E2 -7127.655} C_VEL
LIN {X 0,Y 478.819,Z 515.807,A -85,B 0,C 180,E1 -7128.617,E2 -7128.617} C_VEL
LIN {X 0,Y 479.406,Z 503.721,A -85,B 0,C 180,E1 -7129.37,E2 -7129.37} C_VEL
LIN {X 0,Y 480.095,Z 489.94,A -85,B 0,C 180,E1 -7130.055,E2 -7130.055} C_VEL
LIN {X 0,Y 480.596,Z 474.836,A -85,B 0,C 180,E1 -7130.625,E2 -7130.625} C_VEL
LIN {X 0,Y 480.977,Z 459.373,A -85,B 0,C 180,E1 -7131.024,E2 -7131.024} C_VEL
LIN {X 0,Y 481.887,Z 379.673,A -85,B 0,C 180,E1 -7132.255,E2 -7132.255} C_VEL
LIN {X 0,Y 482.468,Z 314.251,A -85,B 0,C 180,E1 -7133.262,E2 -7133.262} C_VEL
LIN {X 0,Y 478.065,Z 295.144,A -85,B 0,C 180,E1 -7133.819,E2 -7133.819} C_VEL
LIN {X 0,Y 476.479,Z 286.904,A -85,B 0,C 180,E1 -7135.324,E2 -7135.324} C_VEL
LIN {X 0,Y 474.7,Z 278.982,A -85,B 0,C 180,E1 -7136.843,E2 -7136.843} C_VEL
LIN {X 0,Y 474.603,Z 278.993,A -85,B 0,C 180,E1 -7140.229,E2 -7140.229} C_VEL
LIN {X 0,Y 474.64,Z 278.991,A -85,B 0,C 180,E1 -7143.219,E2 -7143.219} C_VEL
LIN {X 0,Y 474.589,Z 278.994,A -85,B 0,C 180,E1 -7146.322,E2 -7146.322} C_VEL
LIN {X 0,Y 474.613,Z 278.988,A -85,B 0,C 180,E1 -7149.645,E2 -7149.645} C_VEL
LIN {X 0,Y 474.609,Z 278.992,A -85,B 0,C 180,E1 -7152.933,E2 -7152.933} C_VEL
LIN {X 0,Y 474.598,Z 278.99,A -85,B 0,C 180,E1 -7155.894,E2 -7155.894} C_VEL
LIN {X 0,Y 474.615,Z 278.983,A -85,B 0,C 180,E1 -7159.041,E2 -7159.041} C_VEL
LIN {X 0,Y 474.602,Z 278.987,A -85,B 0,C 180,E1 -7161.703,E2 -7161.703} C_VEL
LIN {X 0,Y 474.614,Z 278.984,A -85,B 0,C 180,E1 -7164.725,E2 -7164.725} C_VEL
LIN {X 0,Y 474.618,Z 278.982,A -85,B 0,C 180,E1 -7167.786,E2 -7167.786} C_VEL
LIN {X 0,Y 474.612,Z 278.984,A -85,B 0,C 180,E1 -7170.884,E2 -7170.884} C_VEL
LIN {X 0,Y 474.617,Z 278.985,A -85,B 0,C 180,E1 -7173.626,E2 -7173.626} C_VEL
LIN {X 0,Y 474.623,Z 278.989,A -85,B 0,C 180,E1 -7176.641,E2 -7176.641} C_VEL
LIN {X 0,Y 474.641,Z 278.983,A -85,B 0,C 180,E1 -7180.089,E2 -7180.089} C_VEL
LIN {X 0,Y 474.624,Z 278.987,A -85,B 0,C 180,E1 -7182.773,E2 -7182.773} C_VEL
LIN {X 0,Y 474.629,Z 278.984,A -85,B 0,C 180,E1 -7185.42,E2 -7185.42} C_VEL
LIN {X 0,Y 474.691,Z 278.976,A -85,B 0,C 180,E1 -7188.037,E2 -7188.037} C_VEL
LIN {X 0,Y 474.696,Z 278.974,A -85,B 0,C 180,E1 -7191.486,E2 -7191.486} C_VEL
LIN {X 0,Y 474.746,Z 278.97,A -85,B 0,C 180,E1 -7194.052,E2 -7194.052} C_VEL
LIN {X 0,Y 474.869,Z 278.955,A -85,B 0,C 180,E1 -7197.455,E2 -7197.455} C_VEL
LIN {X 0,Y 474.892,Z 278.949,A -85,B 0,C 180,E1 -7200,E2 -7200} C_VEL
LIN {X 0,Y 474.865,Z 278.962,A -85,B 0,C 180,E1 -7202.545,E2 -7202.545} C_VEL
LIN {X 0,Y 474.744,Z 278.97,A -85,B 0,C 180,E1 -7205.948,E2 -7205.948} C_VEL
LIN {X 0,Y 474.685,Z 278.981,A -85,B 0,C 180,E1 -7208.514,E2 -7208.514} C_VEL
LIN {X 0,Y 474.69,Z 278.979,A -85,B 0,C 180,E1 -7211.963,E2 -7211.963} C_VEL
LIN {X 0,Y 474.686,Z 278.978,A -85,B 0,C 180,E1 -7215.456,E2 -7215.456} C_VEL
LIN {X 0,Y 474.648,Z 278.984,A -85,B 0,C 180,E1 -7219.011,E2 -7219.011} C_VEL
LIN {X 0,Y 474.576,Z 278.991,A -85,B 0,C 180,E1 -7221.729,E2 -7221.729} C_VEL
LIN {X 0,Y 474.612,Z 278.991,A -85,B 0,C 180,E1 -7224.495,E2 -7224.495} C_VEL
LIN {X 0,Y 474.626,Z 278.985,A -85,B 0,C 180,E1 -7227.324,E2 -7227.324} C_VEL
LIN {X 0,Y 474.59,Z 278.996,A -85,B 0,C 180,E1 -7230.231,E2 -7230.231} C_VEL
LIN {X 0,Y 474.604,Z 278.984,A -85,B 0,C 180,E1 -7233.223,E2 -7233.223} C_VEL
LIN {X 0,Y 474.56,Z 278.996,A -85,B 0,C 180,E1 -7236.326,E2 -7236.326} C_VEL
LIN {X 0,Y 474.591,Z 278.989,A -85,B 0,C 180,E1 -7239.644,E2 -7239.644} C_VEL
LIN {X 0,Y 474.579,Z 278.995,A -85,B 0,C 180,E1 -7242.232,E2 -7242.232} C_VEL
LIN {X 0,Y 474.608,Z 278.988,A -85,B 0,C 180,E1 -7245.299,E2 -7245.299} C_VEL
LIN {X 0,Y 474.584,Z 278.994,A -85,B 0,C 180,E1 -7248.212,E2 -7248.212} C_VEL
LIN {X 0,Y 474.612,Z 278.989,A -85,B 0,C 180,E1 -7250.452,E2 -7250.452} C_VEL
LIN {X 0,Y 474.575,Z 278.996,A -85,B 0,C 180,E1 -7253.676,E2 -7253.676} C_VEL
LIN {X 0,Y 474.63,Z 278.988,A -85,B 0,C 180,E1 -7256.78,E2 -7256.78} C_VEL
LIN {X 0,Y 474.659,Z 279.019,A -85,B 0,C 180,E1 -7259.928,E2 -7259.928} C_VEL
LIN {X 0,Y 478.57,Z 295.551,A -85,B 0,C 180,E1 -7262.696,E2 -7262.696} C_VEL
LIN {X 0,Y 479.027,Z 299.735,A -85,B 0,C 180,E1 -7263.349,E2 -7263.349} C_VEL
LIN {X 0,Y 477.979,Z 319.834,A -85,B 0,C 180,E1 -7266.237,E2 -7266.237} C_VEL
LIN {X 0,Y 482.453,Z 343.231,A -85,B 0,C 180,E1 -7266.84,E2 -7266.84} C_VEL
LIN {X 0,Y 480.81,Z 486.514,A -85,B 0,C 180,E1 -7269.044,E2 -7269.044} C_VEL
LIN {X 0,Y 480.295,Z 502.43,A -85,B 0,C 180,E1 -7269.47,E2 -7269.47} C_VEL
LIN {X 0,Y 479.685,Z 517.357,A -85,B 0,C 180,E1 -7270.047,E2 -7270.047} C_VEL
LIN {X 0,Y 479.006,Z 530.764,A -85,B 0,C 180,E1 -7270.724,E2 -7270.724} C_VEL
LIN {X 0,Y 478.269,Z 544.275,A -85,B 0,C 180,E1 -7271.583,E2 -7271.583} C_VEL
LIN {X 0,Y 477.423,Z 556.735,A -85,B 0,C 180,E1 -7272.547,E2 -7272.547} C_VEL
LIN {X 0,Y 476.632,Z 569.413,A -85,B 0,C 180,E1 -7273.731,E2 -7273.731} C_VEL
LIN {X 0,Y 475.847,Z 580.932,A -85,B 0,C 180,E1 -7275.021,E2 -7275.021} C_VEL
LIN {X 0,Y 475.302,Z 590.634,A -85,B 0,C 180,E1 -7276.315,E2 -7276.315} C_VEL
LIN {X 0,Y 474.72,Z 599.545,A -85,B 0,C 180,E1 -7277.714,E2 -7277.714} C_VEL
LIN {X 0,Y 474.418,Z 608.105,A -85,B 0,C 180,E1 -7279.329,E2 -7279.329} C_VEL
LIN {X 0,Y 474.052,Z 615.518,A -85,B 0,C 180,E1 -7281.045,E2 -7281.045} C_VEL
LIN {X 0,Y 473.905,Z 621.403,A -85,B 0,C 180,E1 -7282.759,E2 -7282.759} C_VEL
LIN {X 0,Y 473.788,Z 624.899,A -85,B 0,C 180,E1 -7284.04,E2 -7284.04} C_VEL
LIN {X 0,Y 473.701,Z 628.433,A -85,B 0,C 180,E1 -7285.746,E2 -7285.746} C_VEL
LIN {X 0,Y 473.735,Z 630.761,A -85,B 0,C 180,E1 -7287.449,E2 -7287.449} C_VEL
LIN {X 0,Y 473.685,Z 631.93,A -85,B 0,C 180,E1 -7289.15,E2 -7289.15} C_VEL
LIN {X 0,Y 473.685,Z 631.929,A -85,B 0,C 180,E1 -7290.85,E2 -7290.85} C_VEL
LIN {X 0,Y 473.735,Z 630.757,A -85,B 0,C 180,E1 -7292.551,E2 -7292.551} C_VEL
LIN {X 0,Y 473.701,Z 628.429,A -85,B 0,C 180,E1 -7294.254,E2 -7294.254} C_VEL
LIN {X 0,Y 473.781,Z 624.9,A -85,B 0,C 180,E1 -7295.96,E2 -7295.96} C_VEL
LIN {X 0,Y 473.909,Z 620.079,A -85,B 0,C 180,E1 -7297.67,E2 -7297.67} C_VEL
LIN {X 0,Y 474.109,Z 613.834,A -85,B 0,C 180,E1 -7299.384,E2 -7299.384} C_VEL
LIN {X 0,Y 474.539,Z 605.996,A -85,B 0,C 180,E1 -7301.1,E2 -7301.1} C_VEL
LIN {X 0,Y 474.908,Z 597.389,A -85,B 0,C 180,E1 -7302.65,E2 -7302.65} C_VEL
LIN {X 0,Y 475.469,Z 587.615,A -85,B 0,C 180,E1 -7304.116,E2 -7304.116} C_VEL
LIN {X 0,Y 476.088,Z 577.346,A -85,B 0,C 180,E1 -7305.409,E2 -7305.409} C_VEL
LIN {X 0,Y 476.887,Z 565.31,A -85,B 0,C 180,E1 -7306.681,E2 -7306.681} C_VEL
LIN {X 0,Y 477.637,Z 552.844,A -85,B 0,C 180,E1 -7307.777,E2 -7307.777} C_VEL
LIN {X 0,Y 478.526,Z 539.497,A -85,B 0,C 180,E1 -7308.739,E2 -7308.739} C_VEL
LIN {X 0,Y 479.328,Z 524.767,A -85,B 0,C 180,E1 -7309.596,E2 -7309.596} C_VEL
LIN {X 0,Y 480.026,Z 510.068,A -85,B 0,C 180,E1 -7310.255,E2 -7310.255} C_VEL
LIN {X 0,Y 480.52,Z 495.24,A -85,B 0,C 180,E1 -7310.745,E2 -7310.745} C_VEL
LIN {X 0,Y 480.936,Z 480.607,A -85,B 0,C 180,E1 -7311.062,E2 -7311.062} C_VEL
LIN {X 0,Y 482.435,Z 343.132,A -85,B 0,C 180,E1 -7313.161,E2 -7313.161} C_VEL
LIN {X 0,Y 477.962,Z 319.445,A -85,B 0,C 180,E1 -7313.782,E2 -7313.782} C_VEL
LIN {X 0,Y 479.02,Z 299.431,A -85,B 0,C 180,E1 -7316.694,E2 -7316.694} C_VEL
LIN {X 0,Y 478.559,Z 295.534,A -85,B 0,C 180,E1 -7317.305,E2 -7317.305} C_VEL
LIN {X 0,Y 475.196,Z 281.175,A -85,B 0,C 180,E1 -7319.698,E2 -7319.698} C_VEL
LIN {X 0,Y 474.644,Z 278.987,A -85,B 0,C 180,E1 -7320.104,E2 -7320.104} C_VEL
LIN {X 0,Y 474.63,Z 278.986,A -85,B 0,C 180,E1 -7323.22,E2 -7323.22} C_VEL
LIN {X 0,Y 474.575,Z 278.996,A -85,B 0,C 180,E1 -7326.324,E2 -7326.324} C_VEL
LIN {X 0,Y 474.594,Z 278.994,A -85,B 0,C 180,E1 -7329.643,E2 -7329.643} C_VEL
LIN {X 0,Y 474.565,Z 278.994,A -85,B 0,C 180,E1 -7332.938,E2 -7332.938} C_VEL
LIN {X 0,Y 474.594,Z 278.995,A -85,B 0,C 180,E1 -7335.893,E2 -7335.893} C_VEL
LIN {X 0,Y 474.596,Z 278.989,A -85,B 0,C 180,E1 -7339.043,E2 -7339.043} C_VEL
LIN {X 0,Y 474.581,Z 278.996,A -85,B 0,C 180,E1 -7341.707,E2 -7341.707} C_VEL
LIN {X 0,Y 474.601,Z 278.986,A -85,B 0,C 180,E1 -7344.724,E2 -7344.724} C_VEL
LIN {X 0,Y 474.616,Z 278.99,A -85,B 0,C 180,E1 -7347.786,E2 -7347.786} C_VEL
LIN {X 0,Y 474.594,Z 278.988,A -85,B 0,C 180,E1 -7350.888,E2 -7350.888} C_VEL
LIN {X 0,Y 474.569,Z 278.996,A -85,B 0,C 180,E1 -7353.623,E2 -7353.623} C_VEL
LIN {X 0,Y 474.622,Z 278.984,A -85,B 0,C 180,E1 -7356.642,E2 -7356.642} C_VEL
LIN {X 0,Y 474.638,Z 278.975,A -85,B 0,C 180,E1 -7360.089,E2 -7360.089} C_VEL
LIN {X 0,Y 474.613,Z 278.982,A -85,B 0,C 180,E1 -7362.773,E2 -7362.773} C_VEL
LIN {X 0,Y 474.624,Z 278.991,A -85,B 0,C 180,E1 -7365.42,E2 -7365.42} C_VEL
LIN {X 0,Y 474.678,Z 278.964,A -85,B 0,C 180,E1 -7368.037,E2 -7368.037} C_VEL
